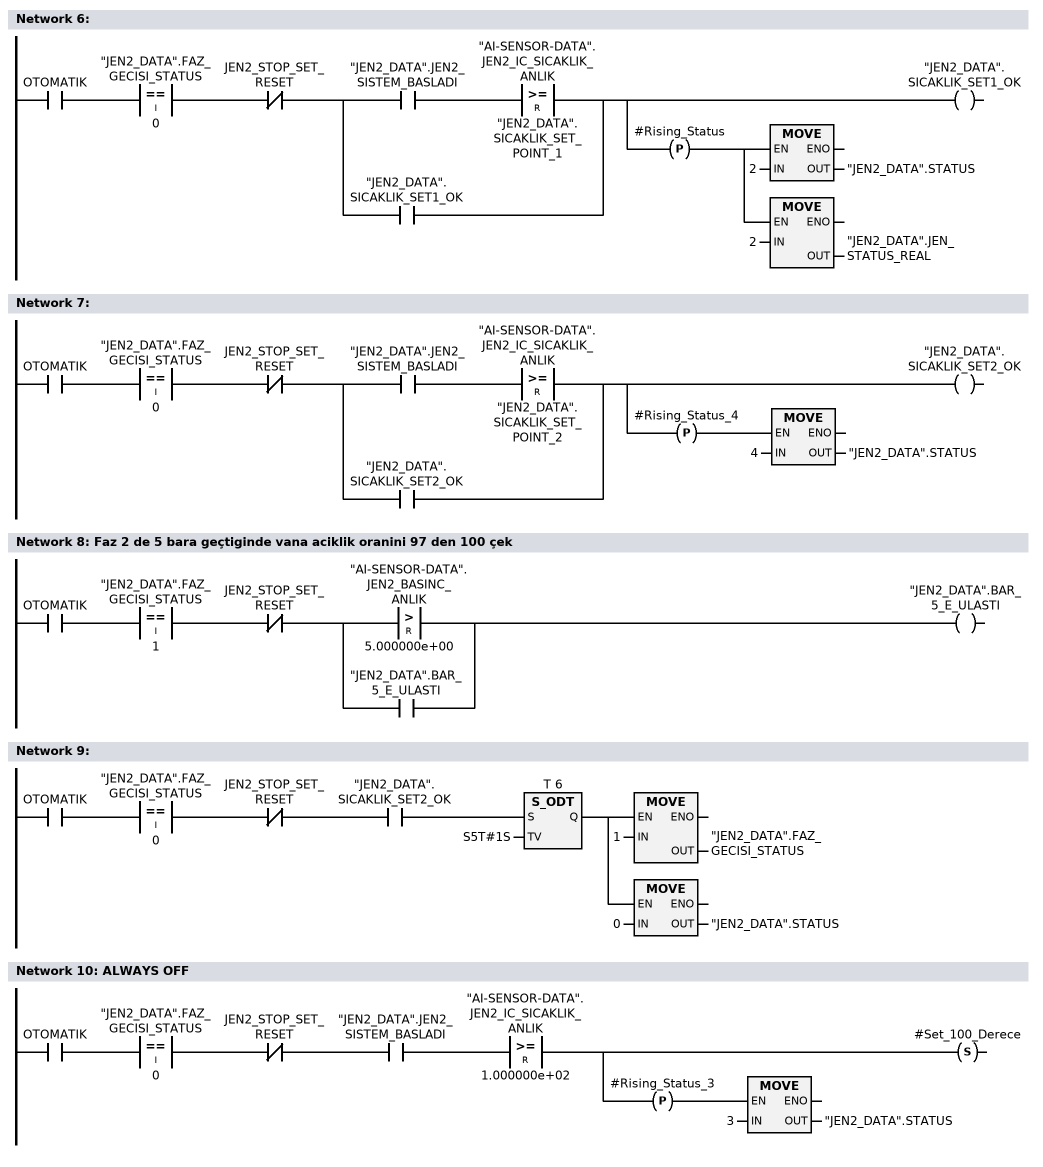
NETWORK
TITLE =
      A     "OTOMATIK";
      A(;
      L     "JEN2_DATA".FAZ_GECISI_STATUS;
      L     0;
      ==I;
      );
      AN    "JEN2_STOP_SET_RESET";
      A(;
      A     "JEN2_DATA".JEN2_SISTEM_BASLADI;
      A(;
      L     "AI-SENSOR-DATA".JEN2_IC_SICAKLIK_ANLIK;
      L     "JEN2_DATA".SICAKLIK_SET_POINT_1;
      >=R;
      );
      O     "JEN2_DATA".SICAKLIK_SET1_OK;
      );
      =     L 0.0;
      A     L 0.0;
      BLD   102;
      =     "JEN2_DATA".SICAKLIK_SET1_OK;
      A     L 0.0;
      FP    #Rising_Status;
      =     L 0.1;
      A     L 0.1;
      JNB   _006;
      L     2;
      T     "JEN2_DATA".STATUS;
_006: NOP   0;
      A     L 0.1;
      JNB   _007;
      L     2;
      T     "JEN2_DATA".JEN_STATUS_REAL;
_007: NOP   0;
NETWORK
TITLE =
      A     "OTOMATIK";
      A(;
      L     "JEN2_DATA".FAZ_GECISI_STATUS;
      L     0;
      ==I;
      );
      AN    "JEN2_STOP_SET_RESET";
      A(;
      A     "JEN2_DATA".JEN2_SISTEM_BASLADI;
      A(;
      L     "AI-SENSOR-DATA".JEN2_IC_SICAKLIK_ANLIK;
      L     "JEN2_DATA".SICAKLIK_SET_POINT_2;
      >=R;
      );
      O     "JEN2_DATA".SICAKLIK_SET2_OK;
      );
      =     L 0.0;
      A     L 0.0;
      BLD   102;
      =     "JEN2_DATA".SICAKLIK_SET2_OK;
      A     L 0.0;
      FP    #Rising_Status_4;
      JNB   _008;
      L     4;
      T     "JEN2_DATA".STATUS;
_008: NOP   0;
NETWORK
TITLE = Faz 2 de 5 bara geçtiginde vana aciklik oranini 97 den 100 çek
      A     "OTOMATIK";
      A(;
      L     "JEN2_DATA".FAZ_GECISI_STATUS;
      L     1;
      ==I;
      );
      AN    "JEN2_STOP_SET_RESET";
      A(;
      O(;
      L     "AI-SENSOR-DATA".JEN2_BASINC_ANLIK;
      L     5.000000e+00;
      >R;
      );
      O     "JEN2_DATA".BAR_5_E_ULASTI;
      );
      =     "JEN2_DATA".BAR_5_E_ULASTI;
NETWORK
TITLE =
//SET 2 SICAKLIGINDAN SONRA FAZ 2 E GEC
      A     "OTOMATIK";
      A(;
      L     "JEN2_DATA".FAZ_GECISI_STATUS;
      L     0;
      ==I;
      );
      AN    "JEN2_STOP_SET_RESET";
      A     "JEN2_DATA".SICAKLIK_SET2_OK;
      L     S5T#1S;
      SD    T 6;
      NOP   0;
      NOP   0;
      NOP   0;
      A     T 6;
      =     L 0.0;
      A     L 0.0;
      JNB   _009;
      L     1;
      T     "JEN2_DATA".FAZ_GECISI_STATUS;
_009: NOP   0;
      A     L 0.0;
      JNB   _00a;
      L     0;
      T     "JEN2_DATA".STATUS;
_00a: NOP   0;
NETWORK
TITLE = ALWAYS OFF
//Pompa 100 derecede duracak
      A     "OTOMATIK";
      A(;
      L     "JEN2_DATA".FAZ_GECISI_STATUS;
      L     0;
      ==I;
      );
      AN    "JEN2_STOP_SET_RESET";
      A     "JEN2_DATA".JEN2_SISTEM_BASLADI;
      A(;
      L     "AI-SENSOR-DATA".JEN2_IC_SICAKLIK_ANLIK;
      L     1.000000e+02;
      >=R;
      );
      =     L 0.0;
      A     L 0.0;
      BLD   102;
      S     #Set_100_Derece;
      A     L 0.0;
      FP    #Rising_Status_3;
      JNB   _00b;
      L     3;
      T     "JEN2_DATA".STATUS;
_00b: NOP   0;
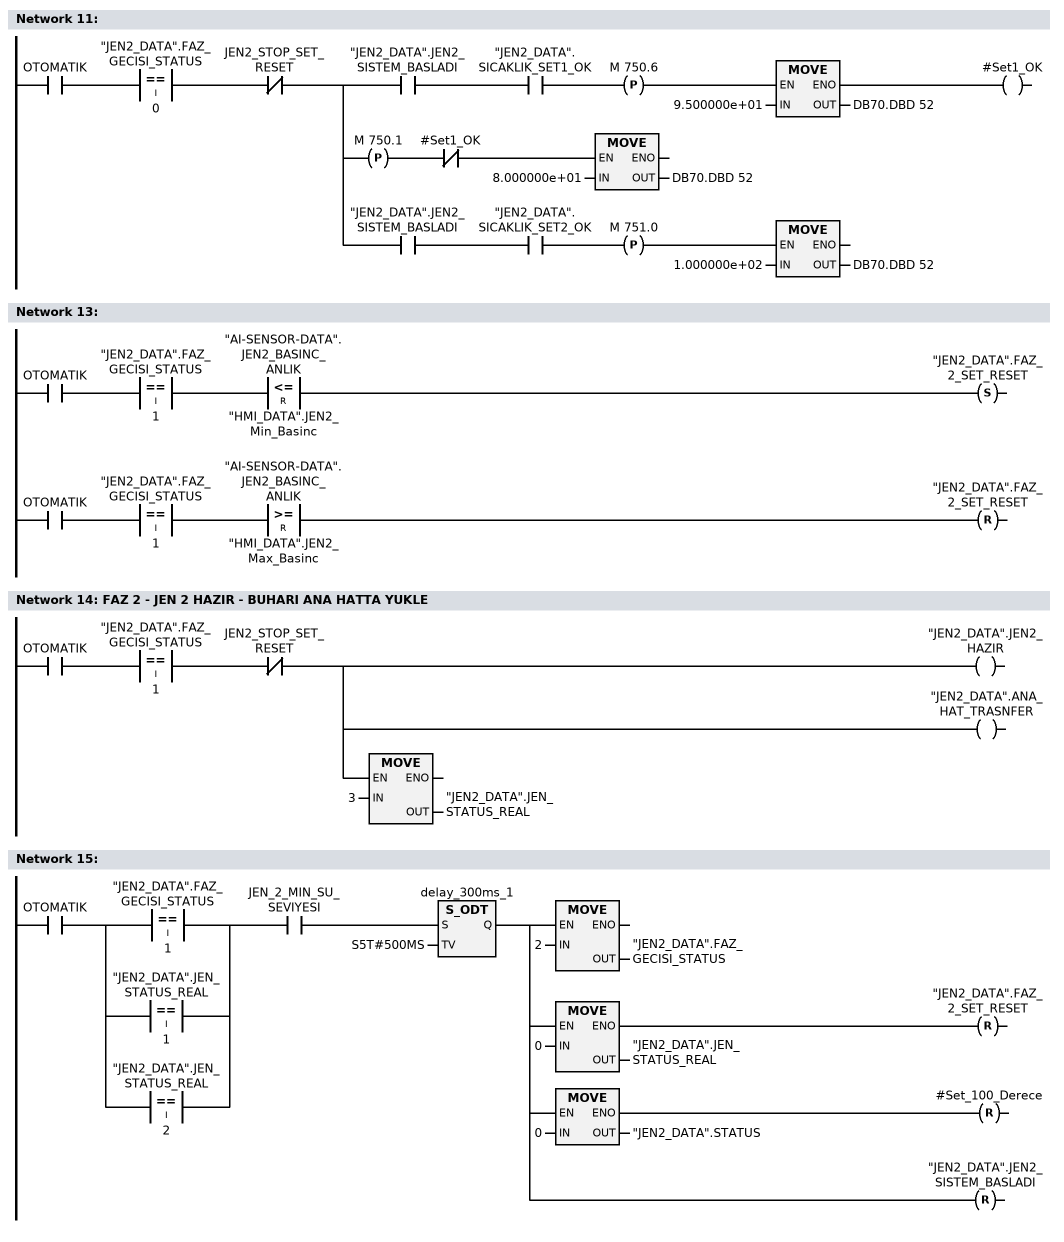
NETWORK
TITLE =
//-Sicaklik set 1 e geldiginde vana kapanma orani 5'e kadar düsüyor
//-Sicaklik set 2 e geldiginde vana kapanma orani 0'a kadar dusecek
      A     "OTOMATIK";
      A(;
      L     "JEN2_DATA".FAZ_GECISI_STATUS;
      L     0;
      ==I;
      );
      AN    "JEN2_STOP_SET_RESET";
      =     L 0.0;
      A     L 0.0;
      A     "JEN2_DATA".JEN2_SISTEM_BASLADI;
      A     "JEN2_DATA".SICAKLIK_SET1_OK;
      FP    M 750.6;
      JNB   _00c;
      L     9.500000e+01;
      T     DB70.DBD 52;
      SET;
      SAVE;
      CLR;
_00c: A     BR;
      =     #Set1_OK;
      A     L 0.0;
      FP    M 750.1;
      AN    #Set1_OK;
      JNB   _00d;
      L     8.000000e+01;
      T     DB70.DBD 52;
_00d: NOP   0;
      A     L 0.0;
      A     "JEN2_DATA".JEN2_SISTEM_BASLADI;
      A     "JEN2_DATA".SICAKLIK_SET2_OK;
      FP    M 751.0;
      JNB   _00e;
      L     1.000000e+02;
      T     DB70.DBD 52;
_00e: NOP   0;
NETWORK
TITLE =
NETWORK
TITLE =
//FAZ - 2 MODUNA GEÇ
//1-BURLOR VE POMPA 4.5-5.5 BAR ARASINDA ÇALISIP DURACAK
      A     "OTOMATIK";
      A(;
      L     "JEN2_DATA".FAZ_GECISI_STATUS;
      L     1;
      ==I;
      );
      A(;
      L     "AI-SENSOR-DATA".JEN2_BASINC_ANLIK;
      L     "HMI_DATA".JEN2_Min_Basinc;
      <=R;
      );
      S     "JEN2_DATA".FAZ_2_SET_RESET;
      A     "OTOMATIK";
      A(;
      L     "JEN2_DATA".FAZ_GECISI_STATUS;
      L     1;
      ==I;
      );
      A(;
      L     "AI-SENSOR-DATA".JEN2_BASINC_ANLIK;
      L     "HMI_DATA".JEN2_Max_Basinc;
      >=R;
      );
      R     "JEN2_DATA".FAZ_2_SET_RESET;
      NOP   0;
NETWORK
TITLE = FAZ 2 - JEN 2 HAZIR - BUHARI ANA HATTA YUKLE
      A     "OTOMATIK";
      A(;
      L     "JEN2_DATA".FAZ_GECISI_STATUS;
      L     1;
      ==I;
      );
      AN    "JEN2_STOP_SET_RESET";
      =     L 0.0;
      A     L 0.0;
      BLD   102;
      =     "JEN2_DATA".JEN2_HAZIR;
      A     L 0.0;
      BLD   102;
      =     "JEN2_DATA".ANA_HAT_TRASNFER;
      A     L 0.0;
      JNB   _00f;
      L     3;
      T     "JEN2_DATA".JEN_STATUS_REAL;
_00f: NOP   0;
NETWORK
TITLE =
//FAZ 3 - GUVENLIK ONLEMLERI 
//1- 6 bar asildiginda -ok
//2- Baca 180 dereceyi gecerse -ok
//3- Su miktari min altina duserse -ok
      A     "OTOMATIK";
      A(;
      O(;
      L     "JEN2_DATA".FAZ_GECISI_STATUS;
      L     1;
      ==I;
      );
      O(;
      L     "JEN2_DATA".JEN_STATUS_REAL;
      L     1;
      ==I;
      );
      O(;
      L     "JEN2_DATA".JEN_STATUS_REAL;
      L     2;
      ==I;
      );
      );
      A     "JEN_2_MIN_SU_SEVIYESI";
      L     S5T#500MS;
      SD    "delay_300ms_1";
      NOP   0;
      NOP   0;
      NOP   0;
      A     "delay_300ms_1";
      =     L 0.0;
      A     L 0.0;
      JNB   _010;
      L     2;
      T     "JEN2_DATA".FAZ_GECISI_STATUS;
_010: NOP   0;
      A     L 0.0;
      JNB   _011;
      L     0;
      T     "JEN2_DATA".JEN_STATUS_REAL;
      SET;
      SAVE;
      CLR;
_011: A     BR;
      R     "JEN2_DATA".FAZ_2_SET_RESET;
      A     L 0.0;
      JNB   _012;
      L     0;
      T     "JEN2_DATA".STATUS;
      SET;
      SAVE;
      CLR;
_012: A     BR;
      R     #Set_100_Derece;
      A     L 0.0;
      BLD   102;
      R     "JEN2_DATA".JEN2_SISTEM_BASLADI;
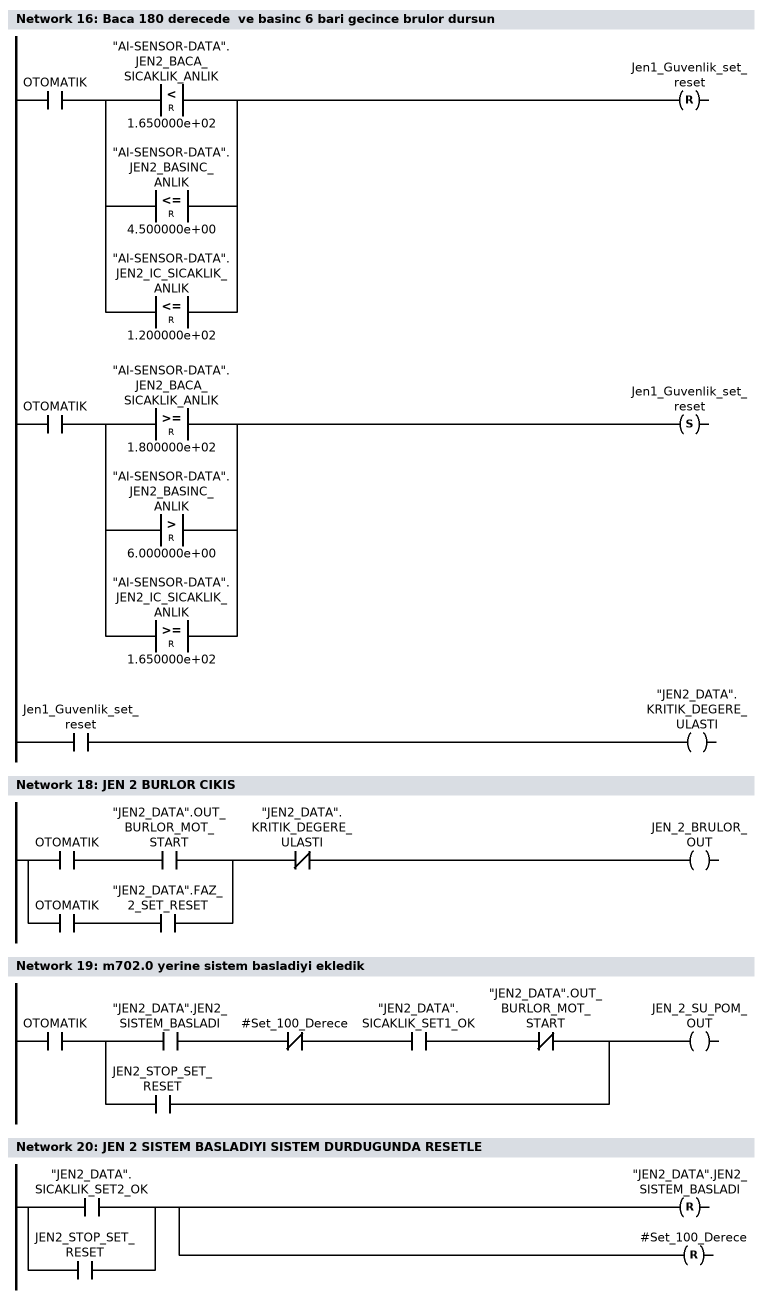
NETWORK
TITLE = Baca 180 derecede  ve basinc 6 bari gecince brulor dursun
      A     "OTOMATIK";
      A(;
      O(;
      L     "AI-SENSOR-DATA".JEN2_BACA_SICAKLIK_ANLIK;
      L     1.650000e+02;
      <R;
      );
      O(;
      L     "AI-SENSOR-DATA".JEN2_BASINC_ANLIK;
      L     4.500000e+00;
      <=R;
      );
      O(;
      L     "AI-SENSOR-DATA".JEN2_IC_SICAKLIK_ANLIK;
      L     1.200000e+02;
      <=R;
      );
      );
      R     "Jen1_Guvenlik_set_reset";
      A     "OTOMATIK";
      A(;
      O(;
      L     "AI-SENSOR-DATA".JEN2_BACA_SICAKLIK_ANLIK;
      L     1.800000e+02;
      >=R;
      );
      O(;
      L     "AI-SENSOR-DATA".JEN2_BASINC_ANLIK;
      L     6.000000e+00;
      >R;
      );
      O(;
      L     "AI-SENSOR-DATA".JEN2_IC_SICAKLIK_ANLIK;
      L     1.650000e+02;
      >=R;
      );
      );
      S     "Jen1_Guvenlik_set_reset";
      A     "Jen1_Guvenlik_set_reset";
      =     "JEN2_DATA".KRITIK_DEGERE_ULASTI;
NETWORK
TITLE =
NETWORK
TITLE = JEN 2 BURLOR CIKIS
      A(;
      A     "OTOMATIK";
      A     "JEN2_DATA".OUT_BURLOR_MOT_START;
      O;
      A     "OTOMATIK";
      A     "JEN2_DATA".FAZ_2_SET_RESET;
      );
      AN    "JEN2_DATA".KRITIK_DEGERE_ULASTI;
      =     "JEN_2_BRULOR_OUT";
NETWORK
TITLE = m702.0 yerine sistem basladiyi ekledik
      A     "OTOMATIK";
      A(;
      A     "JEN2_DATA".JEN2_SISTEM_BASLADI;
      AN    #Set_100_Derece;
      A     "JEN2_DATA".SICAKLIK_SET1_OK;
      AN    "JEN2_DATA".OUT_BURLOR_MOT_START;
      O     "JEN2_STOP_SET_RESET";
      );
      =     "JEN_2_SU_POM_OUT";
NETWORK
TITLE = JEN 2 SISTEM BASLADIYI SISTEM DURDUGUNDA RESETLE
      O     "JEN2_DATA".SICAKLIK_SET2_OK;
      O     "JEN2_STOP_SET_RESET";
      R     "JEN2_DATA".JEN2_SISTEM_BASLADI;
      R     #Set_100_Derece;
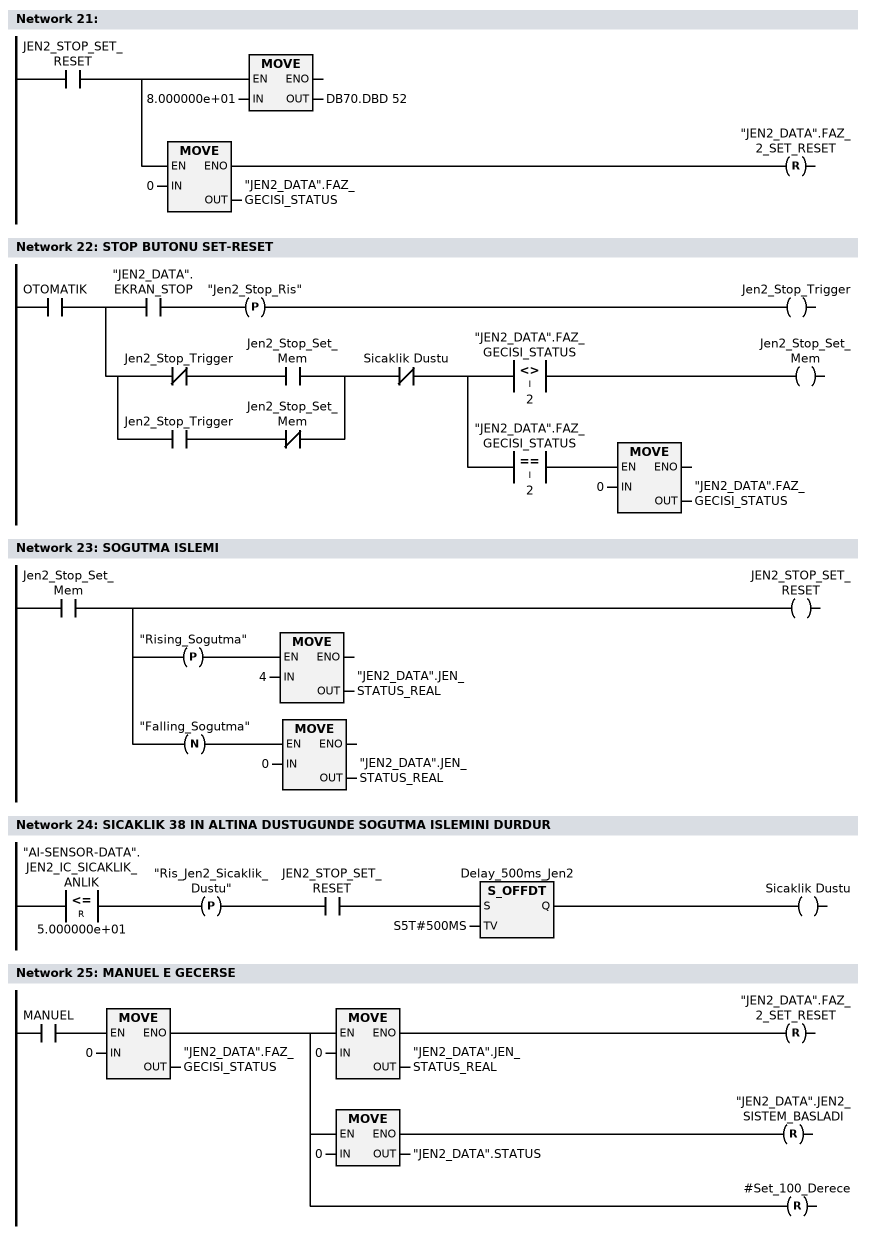
NETWORK
TITLE =
      A     "JEN2_STOP_SET_RESET";
      =     L 0.0;
      A     L 0.0;
      JNB   _013;
      L     8.000000e+01;
      T     DB70.DBD 52;
_013: NOP   0;
      A     L 0.0;
      JNB   _014;
      L     0;
      T     "JEN2_DATA".FAZ_GECISI_STATUS;
      SET;
      SAVE;
      CLR;
_014: A     BR;
      R     "JEN2_DATA".FAZ_2_SET_RESET;
NETWORK
TITLE = STOP BUTONU SET-RESET
      A     "OTOMATIK";
      =     L 0.0;
      A     L 0.0;
      A     "JEN2_DATA".EKRAN_STOP;
      FP    "Jen2_Stop_Ris";
      =     "Jen2_Stop_Trigger";
      A     L 0.0;
      A(;
      AN    "Jen2_Stop_Trigger";
      A     "Jen2_Stop_Set_Mem";
      O;
      A     "Jen2_Stop_Trigger";
      AN    "Jen2_Stop_Set_Mem";
      );
      AN    "Sicaklik Dustu";
      =     L 0.1;
      A     L 0.1;
      A(;
      L     "JEN2_DATA".FAZ_GECISI_STATUS;
      L     2;
      <>I;
      );
      =     "Jen2_Stop_Set_Mem";
      A     L 0.1;
      A(;
      L     "JEN2_DATA".FAZ_GECISI_STATUS;
      L     2;
      ==I;
      );
      JNB   _015;
      L     0;
      T     "JEN2_DATA".FAZ_GECISI_STATUS;
_015: NOP   0;
NETWORK
TITLE = SOGUTMA ISLEMI
      A     "Jen2_Stop_Set_Mem";
      =     L 0.0;
      A     L 0.0;
      BLD   102;
      =     "JEN2_STOP_SET_RESET";
      A     L 0.0;
      FP    "Rising_Sogutma";
      JNB   _016;
      L     4;
      T     "JEN2_DATA".JEN_STATUS_REAL;
_016: NOP   0;
      A     L 0.0;
      FN    "Falling_Sogutma";
      JNB   _017;
      L     0;
      T     "JEN2_DATA".JEN_STATUS_REAL;
_017: NOP   0;
NETWORK
TITLE = SICAKLIK 38 IN ALTINA DUSTUGUNDE SOGUTMA ISLEMINI DURDUR
      A(;
      L     "AI-SENSOR-DATA".JEN2_IC_SICAKLIK_ANLIK;
      L     5.000000e+01;
      <=R;
      );
      FP    "Ris_Jen2_Sicaklik_Dustu";
      A     "JEN2_STOP_SET_RESET";
      L     S5T#500MS;
      SF    "Delay_500ms_Jen2";
      NOP   0;
      NOP   0;
      NOP   0;
      A     "Delay_500ms_Jen2";
      =     "Sicaklik Dustu";
NETWORK
TITLE = MANUEL E GECERSE
      A     "MANUEL";
      JNB   _018;
      L     0;
      T     "JEN2_DATA".FAZ_GECISI_STATUS;
      SET;
      SAVE;
      CLR;
_018: A     BR;
      =     L 0.0;
      A     L 0.0;
      JNB   _019;
      L     0;
      T     "JEN2_DATA".JEN_STATUS_REAL;
      SET;
      SAVE;
      CLR;
_019: A     BR;
      R     "JEN2_DATA".FAZ_2_SET_RESET;
      A     L 0.0;
      JNB   _01a;
      L     0;
      T     "JEN2_DATA".STATUS;
      SET;
      SAVE;
      CLR;
_01a: A     BR;
      R     "JEN2_DATA".JEN2_SISTEM_BASLADI;
      A     L 0.0;
      BLD   102;
      R     #Set_100_Derece;
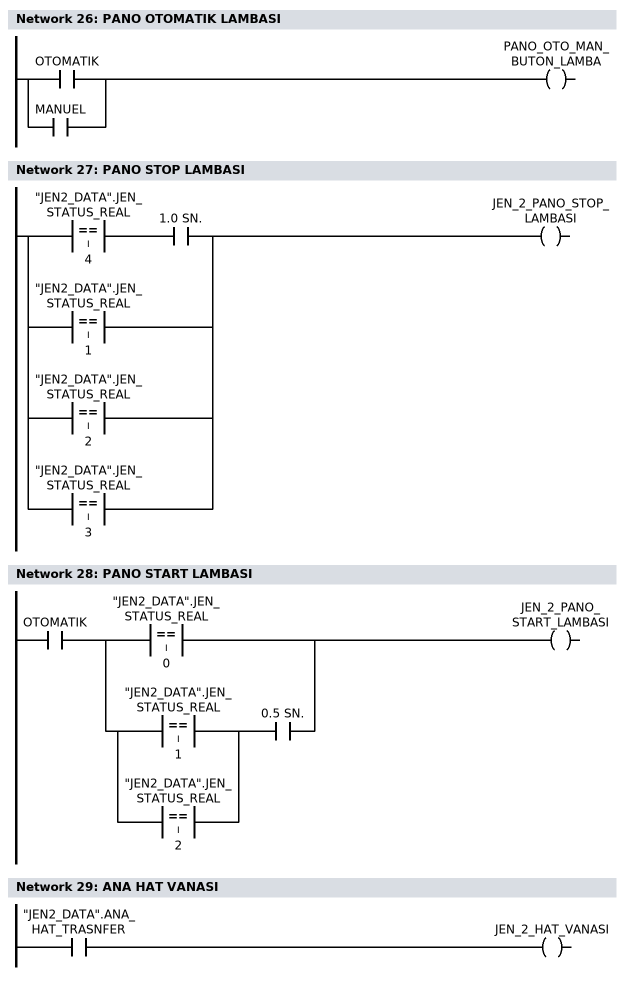
NETWORK
TITLE = PANO OTOMATIK LAMBASI
      O     "OTOMATIK";
      O     "MANUEL";
      =     "PANO_OTO_MAN_BUTON_LAMBA";
NETWORK
TITLE = PANO STOP LAMBASI
//1- Buhar hazýrlaniyor
//2- set 1 e ulasti
//3- Basinci Stabil tutma
//4- Sogutma
      A(;
      L     "JEN2_DATA".JEN_STATUS_REAL;
      L     4;
      ==I;
      );
      A     "1.0 SN.";
      O(;
      L     "JEN2_DATA".JEN_STATUS_REAL;
      L     1;
      ==I;
      );
      O(;
      L     "JEN2_DATA".JEN_STATUS_REAL;
      L     2;
      ==I;
      );
      O(;
      L     "JEN2_DATA".JEN_STATUS_REAL;
      L     3;
      ==I;
      );
      =     "JEN_2_PANO_STOP_LAMBASI";
NETWORK
TITLE = PANO START LAMBASI
      A     "OTOMATIK";
      A(;
      O(;
      L     "JEN2_DATA".JEN_STATUS_REAL;
      L     0;
      ==I;
      );
      O;
      A(;
      O(;
      L     "JEN2_DATA".JEN_STATUS_REAL;
      L     1;
      ==I;
      );
      O(;
      L     "JEN2_DATA".JEN_STATUS_REAL;
      L     2;
      ==I;
      );
      );
      A     "0.5 SN.";
      );
      =     "JEN_2_PANO_START_LAMBASI";
NETWORK
TITLE = ANA HAT VANASI 
      A     "JEN2_DATA".ANA_HAT_TRASNFER;
      =     "JEN_2_HAT_VANASI";
END_FUNCTION_BLOCK

FUNCTION "TIME_UNSCALE" : VOID	// FC 1
VERSION : 0.0
VAR_INPUT
  iTimeET : TIME ;
  iIstenileSure : S5TIME ;
END_VAR
VAR_OUTPUT
  oOUT : DINT ;
END_VAR
VAR_TEMP
  vTemp : DINT ;
  vValue : DINT ;
  vValue2 : DINT ;
  vIstenilenTime : TIME ;
  vIstenilenDint : DINT ;
END_VAR
BEGIN
// body was compiled from an SCL source; compiled code not shown
END_FUNCTION

FUNCTION "O.Vana_AciklikHesaplama" : VOID	// FC 2
VERSION : 0.1
VAR_INPUT
  IlkAciklikDegeri : REAL ;
  KademeliAcikDegeri : REAL ;
END_VAR
VAR_OUTPUT
  oKademe_1 : REAL ;
  oKademe_2 : REAL ;
  oKademe_3 : REAL ;
  oKademe_4 : REAL ;
  oKademe_5 : REAL ;
  oKademe_6 : REAL ;
  oKademe_7 : REAL ;
END_VAR
VAR_TEMP
  tKademe : STRUCT
   Iki : REAL ;
   Uc : REAL ;
   Dort : REAL ;
   Bes : REAL ;
   Alti : REAL ;
   Yedi : REAL ;
  END_STRUCT ;
  tCheck_Kademe5 : BOOL ;
  tCheck_Kademe6 : BOOL ;
  tCheck_Kademe7 : BOOL ;
END_VAR
BEGIN
NETWORK
TITLE =
//------------------------
// kademe 1
      L     #IlkAciklikDegeri;
      T     #oKademe_1;
//------------------------
// kademe 2
      L     #IlkAciklikDegeri;
      L     #KademeliAcikDegeri;
      +R;
      T     #tKademe.Iki;
      L     #tKademe.Iki;
      T     #oKademe_2;
//-----------------------
// kademe 3
      L     #KademeliAcikDegeri;
      L     #tKademe.Iki;
      +R;
      T     #tKademe.Uc;
      L     #tKademe.Uc;
      T     #oKademe_3;
//-----------------------
// kademe 4
      L     #KademeliAcikDegeri;
      L     #tKademe.Uc;
      +R;
      T     #tKademe.Dort;
      L     #tKademe.Dort;
      T     #oKademe_4;
//-----------------------
// kademe 5
      L     #KademeliAcikDegeri;
      L     #tKademe.Dort;
      +R;
      T     #tKademe.Bes;
      L     #tKademe.Bes;
      L     6.000000e+01;
      >R;
      =     #tCheck_Kademe5;
      A     #tCheck_Kademe5;
      JNB   j005;
      L     6.000000e+01;
      T     #tKademe.Bes;
j005: NOP   0;
      L     #tKademe.Bes;
      T     #oKademe_5;
//-----------------------
// kademe 6
      L     #KademeliAcikDegeri;
      L     #tKademe.Bes;
      +R;
      T     #tKademe.Alti;
      L     #tKademe.Alti;
      L     6.000000e+01;
      >R;
      =     #tCheck_Kademe6;
      A     #tCheck_Kademe6;
      JNB   j006;
      L     6.000000e+01;
      T     #tKademe.Alti;
j006: NOP   0;
      L     #tKademe.Alti;
      T     #oKademe_6;
//-----------------------
// kademe 7
      L     #KademeliAcikDegeri;
      L     #tKademe.Alti;
      +R;
      T     #tKademe.Yedi;
      L     #tKademe.Yedi;
      L     6.000000e+01;
      >R;
      =     #tCheck_Kademe7;
      A     #tCheck_Kademe7;
      JNB   j007;
      L     6.000000e+01;
      T     #tKademe.Yedi;
j007: NOP   0;
      L     #tKademe.Yedi;
      T     #oKademe_7;
NETWORK
TITLE =
END_FUNCTION

FUNCTION "IntToS5Time" : VOID	// FC 10
VERSION : 0.0
VAR_INPUT
  Saat : INT ;
  Dakika : INT ;
END_VAR
VAR_OUTPUT
  HesaplananSure_S5TIME : S5TIME ;
END_VAR
VAR_TEMP
  tSaat_Dint : DINT ;
  tHesaplananSaat : DINT ;
  tDakika_Dint : DINT ;
  tHesaplananDakika : DINT ;
  tHesaplnananSure_Dint : DINT ;
  tHesaplananSure_Time : TIME ;
END_VAR
BEGIN
// body was compiled from an SCL source; compiled code not shown
END_FUNCTION

// FC 33: know-how protected block, not included

// FC 40: know-how protected block, not included

// FC 105: know-how protected block, not included

// FC 106: know-how protected block, not included

DATA_BLOCK "AI-SENSOR-DATA"	// DB 1
VERSION : 0.1
  STRUCT
   JEN1_BASINC_ANLIK : REAL ;
   JEN2_BASINC_ANLIK : REAL ;
   JEN1_BASINC_RET_VAL : WORD ;
   JEN2_BASINC_RET_VAL : WORD ;
   JEN1_IC_SICAKLIK_ANLIK : REAL ;
   JEN2_IC_SICAKLIK_ANLIK : REAL ;
   JEN1_IC_SICAKLIK_RET_VAL : WORD ;
   JEN2_IC_SICAKLIK_RET_VAL : WORD ;
   JEN1_BACA_SICAKLIK_ANLIK : REAL ;
   JEN2_BACA_SICAKLIK_ANLIK : REAL ;
   JEN1_BACA_SICAKLIK_RET_V : WORD ;
   JEN2_BACA_SICAKLIK_RET_V : WORD ;
   HAT_BASINCI_RET_V : WORD ;
   HAT_BASINCI_ANLIK : REAL ;
   HAVA_BASINCI_RET_V : WORD ;
   HAVA_BASINCI_ANLIK : REAL ;
   HAT_BASINCI_YETERLI : BOOL ;
  END_STRUCT ;	
BEGIN
END_DATA_BLOCK

DATA_BLOCK "ORTAK_DATA"	// DB 2
VERSION : 0.1
  STRUCT
   JEN_EMNIYET_BASINCI : REAL ;
   JEN_EMNIYET_SICAKLIGI : REAL ;
   OTO_EMNIYET_BASINCI : REAL ;
   OTO_EMNIYET_SICAKLIGI : REAL ;
   OTO_ISLEM_BITTI_VANA_AC : BOOL ;
   OTO_JEN_DURDU : REAL ;
  END_STRUCT ;	
BEGIN
END_DATA_BLOCK

DATA_BLOCK "TIME_OTO_1_DB"	// DB 5
AUTHOR : SIMATIC
FAMILY : IEC_TC
VERSION : 0.0
"TON"
BEGIN
END_DATA_BLOCK

DATA_BLOCK "TIME_OTO_2_DB"	// DB 6
AUTHOR : SIMATIC
FAMILY : IEC_TC
VERSION : 0.0
"TON"
BEGIN
END_DATA_BLOCK

DATA_BLOCK "TIME_OTO_1_PROSES_DB"	// DB 7
AUTHOR : SIMATIC
FAMILY : IEC_TC
VERSION : 0.0
"TON"
BEGIN
END_DATA_BLOCK

DATA_BLOCK "TIME_OTO_2_PROSES_DB"	// DB 8
AUTHOR : SIMATIC
FAMILY : IEC_TC
VERSION : 0.0
"TON"
BEGIN
END_DATA_BLOCK

DATA_BLOCK DB 9
AUTHOR : SIMATIC
FAMILY : IEC_TC
VERSION : 0.0
"TON"
BEGIN
END_DATA_BLOCK

DATA_BLOCK DB 10
AUTHOR : SIMATIC
FAMILY : IEC_TC
VERSION : 0.0
"TON"
BEGIN
END_DATA_BLOCK

DATA_BLOCK "SURELER_DB"	// DB 14
VERSION : 0.0
"SURELER"
BEGIN
END_DATA_BLOCK

DATA_BLOCK "SAFETY_DB"	// DB 15
VERSION : 0.0
"SAFETY"
BEGIN
END_DATA_BLOCK

DATA_BLOCK "KAZAN1_DATA"	// DB 17
VERSION : 0.1
  STRUCT
   IN_STATUS : INT ;
   IN_JEN_OK : BOOL ;
   IN_DIGER_KAZ_TRANS_HAZIR : BOOL ;
   IN_PISIM_SURESI : S5TIME ;
   IN_SCALE_BASINC_PER : INT ;
   IN_SET_BASINC : REAL ;
   IN_DIGER_KAZAN_BASINCI : REAL ;
   O_PID_MAN_ON : BOOL ;
   O_PID_MAN : REAL ;
   O_TRANSFER_YAPILIYOR : BOOL ;
   O_SCALE_BASINC_RET_VAL : WORD ;
   O_SCALE_BASINC_OUT : REAL ;
   O_TRANSFERE_HAZIR : BOOL ;
   O_SCALE_SICAKLIK_RET_VAL : WORD ;
   O_SCALE_SICAKLIK_OUT : REAL ;
   IN_SCALE_SICAKLIK_PER : INT ;
   O_KAZAN_BOSALTIMDA : BOOL ;
   IN_DIGER_KAZ_BOSALTIMDA : BOOL ;
   IN_DIGER_KAZ_TRANSFERDE : BOOL ;
   O_PISIM_BASLADI : BOOL ;
   PISIM_GECEN_SURE_TIME : TIME ;
   PISIM_GECEN_SURE_DINT : DINT ;
   PROSES_SURESI_TIME : TIME ;
   PROSES_SURESI_DINT : DINT ;
   BEKLEME_SURESI_TIME : TIME ;
   BEKLEME_SURESI_DINT : DINT ;
  END_STRUCT ;	
BEGIN
END_DATA_BLOCK

DATA_BLOCK "KAZAN2_DATA"	// DB 18
VERSION : 0.1
  STRUCT
   IN_STATUS : INT ;
   IN_JEN_OK : BOOL ;
   IN_DIGER_KAZ_TRANS_HAZIR : BOOL ;
   IN_PISIM_SURESI : S5TIME ;
   IN_SCALE_BASINC_PER : INT ;
   IN_SET_BASINC : REAL ;
   IN_DIGER_KAZAN_BASINCI : REAL ;
   O_PID_MAN_ON : BOOL ;
   O_PID_MAN : REAL ;
   O_TRANSFER_YAPILIYOR : BOOL ;
   O_SCALE_BASINC_RET_VAL : WORD ;
   O_SCALE_BASINC_OUT : REAL ;
   O_TRANSFERE_HAZIR : BOOL ;
   O_SCALE_SICAKLIK_RET_VAL : WORD ;
   O_SCALE_SICAKLIK_OUT : REAL ;
   IN_SCALE_SICAKLIK_PER : INT ;
   O_KAZAN_BOSALTIMDA : BOOL ;
   IN_DIGER_KAZ_BOSALTIMDA : BOOL ;
   IN_DIGER_KAZ_TRANSFERDE : BOOL ;
   O_PISIM_BASLADI : BOOL ;
   PISIM_GECEN_SURE_TIME : TIME ;
   PISIM_GECEN_SURE_DINT : DINT ;
   PROSES_SURESI_TIM : TIME ;
   PROSES_SURESI_DINT : DINT ;
   BEKLEME_SURESI_TIME : TIME ;
   BEKLEME_SURESI_DINT : DINT ;
  END_STRUCT ;	
BEGIN
END_DATA_BLOCK

DATA_BLOCK "JEN1_DATA"	// DB 19
VERSION : 0.1
  STRUCT
   BASINC_SET_POINT : REAL ;
   STATUS : INT ;
   SICAKLIK_SET_POINT_1 : REAL ;
   SICAKLIK_SET_POINT_2 : REAL ;
   SISTEM_BASLADI : BOOL ;
   EKRAN_START : BOOL ;
   EKRAN_STOP : BOOL ;
   OUT_BURLOR_MOT_START : BOOL ;
   SICAKLIK_SET1_OK : BOOL ;
   SICAKLIK_SET2_OK : BOOL ;
   OUT_PID_START : BOOL ;
   FAZ_GECISI_STATUS : INT ;
   FAZ_2_SET_RESET : BOOL ;
   BAR_5_E_ULASTI : BOOL ;
   JEN1_HAZIR : BOOL ;
   ANA_HAT_TRASFER_HAZIR : BOOL ;
   JEN_STATUS_REAL : INT ;
   STOP_SET_RESET : BOOL ;
   CALISMA_SURESI_TIME : TIME ;
   CALISMA_SURESI_DINT : DINT ;
   KRITIK_DEGERLERE_ULASTI : BOOL ;	//180 derece baca-6 bari gecti- 165 ic sicaklik
   CALISMA_SURESI_EKRAN : DINT ;
   SET2_DEGERINE_ULASMADI : BOOL ;
  END_STRUCT ;	
BEGIN
END_DATA_BLOCK

DATA_BLOCK "JEN2_DATA"	// DB 20
VERSION : 0.1
  STRUCT
   BASINC_SET_POINT : REAL ;
   STATUS : INT ;
   SICAKLIK_SET_POINT_1 : REAL ;
   SICAKLIK_SET_POINT_2 : REAL ;
   JEN2_SISTEM_BASLADI : BOOL ;
   EKRAN_START : BOOL ;
   EKRAN_STOP : BOOL ;
   OUT_BURLOR_MOT_START : BOOL ;
   SICAKLIK_SET1_OK : BOOL ;
   SICAKLIK_SET2_OK : BOOL ;
   OUT_PID_START : BOOL ;
   FAZ_GECISI_STATUS : INT ;
   FAZ_2_SET_RESET : BOOL ;
   BAR_5_E_ULASTI : BOOL ;
   JEN2_HAZIR : BOOL ;
   ANA_HAT_TRASNFER : BOOL ;
   JEN_STATUS_REAL : INT ;
   STOP_SET_RESET : BOOL ;
   CALISMA_SURESI_TIME : TIME ;
   CALISMA_SURESI_DINT : DINT ;
   KRITIK_DEGERE_ULASTI : BOOL ;	//Baca 180 derecede-6 bari gecti-165 ic sicaklik
   CALISMA_SURESI_EKRAN : DINT ;
  END_STRUCT ;	
BEGIN
END_DATA_BLOCK

DATA_BLOCK "JEN1_PID_DATA"	// DB 21
VERSION : 0.1
  STRUCT
   TCONT_C_LMN : REAL ;
   TCONT_C_LMN_PER : INT ;
  END_STRUCT ;	
BEGIN
END_DATA_BLOCK

DATA_BLOCK "JEN2_PID_DATA"	// DB 22
VERSION : 0.1
  STRUCT
   TCONT_C_LMN : REAL ;
   TCONT_C_LMN_PER : INT ;
  END_STRUCT ;	
BEGIN
END_DATA_BLOCK

DATA_BLOCK "KAZAN1_PID_DATA"	// DB 23
VERSION : 0.1
  STRUCT
   TCONT_LMN_PER : INT ;
   TCONT_LMN : REAL ;
  END_STRUCT ;	
BEGIN
END_DATA_BLOCK

DATA_BLOCK "KAZAN2_PID_DATA"	// DB 24
VERSION : 0.1
  STRUCT
   TCONT_LMN_PER : INT ;
   TCONT_LMN : REAL ;
  END_STRUCT ;	
BEGIN
END_DATA_BLOCK

DATA_BLOCK DB 50
AUTHOR : SIMATIC
FAMILY : ICONT
VERSION : 0.0
"CONT_C"
BEGIN
END_DATA_BLOCK

DATA_BLOCK "JEN2_KONTROL_BLOGU_DB"	// DB 51
VERSION : 0.0
"JEN2_PID_KONTROL"
BEGIN
END_DATA_BLOCK

DATA_BLOCK DB 52
VERSION : 0.0
"JEN1_PID_KONTROL"
BEGIN
END_DATA_BLOCK

DATA_BLOCK "JEN_1_PID_DB"	// DB 69
AUTHOR : SIMATIC
FAMILY : CONTROL
VERSION : 0.0
"TCONT_CP"
BEGIN
END_DATA_BLOCK

DATA_BLOCK "JEN_2_PID_DB"	// DB 70
AUTHOR : SIMATIC
FAMILY : CONTROL
VERSION : 0.0
"TCONT_CP"
BEGIN
END_DATA_BLOCK

DATA_BLOCK "OTOKLAV_1_DB"	// DB 94
VERSION : 0.0
"KAZAN_1_KONTROL"
BEGIN
END_DATA_BLOCK

DATA_BLOCK "OTOKLAV_2_DB"	// DB 95
VERSION : 0.0
"KAZAN_2_KONTROL"
BEGIN
END_DATA_BLOCK

DATA_BLOCK "FB98_DB"	// DB 98
VERSION : 0.0
"JEN1_KONTROL_BLOGU"
BEGIN
END_DATA_BLOCK

DATA_BLOCK "FB99_DB"	// DB 99
VERSION : 0.0
"JEN2_KONTROL_BLOGU"
BEGIN
END_DATA_BLOCK

DATA_BLOCK "HMI_DATA"	// DB 100
VERSION : 0.1
  STRUCT
   JEN1_Min_Basinc : REAL  := 5.000000e+000;	//Jenerator 1 min otomatik sekans basinci
   JEN1_Max_Basinc : REAL  := 5.500000e+000;	//Jenerator 1 max otomatik sekans basinci
   JEN2_Min_Basinc : REAL  := 5.000000e+000;	//Jenerator 2 min otomatik sekans basinci
   JEN2_Max_Basinc : REAL  := 5.500000e+000;	//Jenerator 2 max otomatik sekans basinci
   OTOKLAV_First_Oran : REAL  := 2.000000e+001;	//Otoklav oransal vana otomatik sekans ilk acilis orani
   OTOKLAV_Kademeli_Artis : REAL  := 5.000000e+000;	//Otoklav oransal vana kademeli artis katsayisi
   Otoklav_1_TimeData : STRUCT 	//Otoklav 1 hmi süre bilgisi
    Hours : INT ;	//Istenen calisma saati
    Minutes : INT  := 30;	//Istenen calisma dakikasi
    Second : INT ;	//Istenen calisma saniyesi
   END_STRUCT ;
   Otoklav_2_TimeData : STRUCT 	//Otoklav 2 hmi süre bilgisi
    Hours : INT ;	//Istenen calisma saati
    Minutes : INT  := 30;	//Istenen calisma dakikasi
    Second : INT ;	//Istenen calisma saniyesi
   END_STRUCT ;
  END_STRUCT ;	
BEGIN
   JEN1_Min_Basinc := 5.000000e+00;
   JEN1_Max_Basinc := 5.500000e+00;
   JEN2_Min_Basinc := 5.000000e+00;
   JEN2_Max_Basinc := 5.500000e+00;
   Otoklav_1_TimeData.Minutes := 30;
   Otoklav_2_TimeData.Minutes := 30;
END_DATA_BLOCK

DATA_BLOCK DB 120
VERSION : 0.0
"KAZAN_ORTAK"
BEGIN
END_DATA_BLOCK

DATA_BLOCK "KAZAN_1_PID_DB"	// DB 130
AUTHOR : SIMATIC
FAMILY : CONTROL
VERSION : 0.0
"TCONT_CP"
BEGIN
END_DATA_BLOCK

DATA_BLOCK DB 131
VERSION : 0.0
"KAZAN_1_PID_KONTROL"
BEGIN
END_DATA_BLOCK

DATA_BLOCK DB 132
VERSION : 0.0
"KAZAN_2_PID_KONTROL"
BEGIN
END_DATA_BLOCK

DATA_BLOCK DB 230
VERSION : 0.0
"KAZAN_ORTAK"
BEGIN
END_DATA_BLOCK

DATA_BLOCK "KAZAN_2_PID_DATA"	// DB 231
AUTHOR : SIMATIC
FAMILY : CONTROL
VERSION : 0.0
"TCONT_CP"
BEGIN
END_DATA_BLOCK

DATA_BLOCK DB 232
VERSION : 0.0
"TEST_BLOGU"
BEGIN
END_DATA_BLOCK

ORGANIZATION_BLOCK OB 1
TITLE = "Main Program Sweep (Cycle)"
VERSION : 0.1
VAR_TEMP
  OB1_EV_CLASS : BYTE ;	//Bits 0-3 = 1 (Coming event), Bits 4-7 = 1 (Event class 1)
  OB1_SCAN_1 : BYTE ;	//1 (Cold restart scan 1 of OB 1), 3 (Scan 2-n of OB 1)
  OB1_PRIORITY : BYTE ;	//Priority of OB Execution
  OB1_OB_NUMBR : BYTE ;	//1 (Organization block 1, OB1)
  OB1_RESERVED_1 : BYTE ;	//Reserved for system
  OB1_RESERVED_2 : BYTE ;	//Reserved for system
  OB1_PREV_CYCLE : INT ;	//Cycle time of previous OB1 scan (milliseconds)
  OB1_MIN_CYCLE : INT ;	//Minimum cycle time of OB1 (milliseconds)
  OB1_MAX_CYCLE : INT ;	//Maximum cycle time of OB1 (milliseconds)
  OB1_DATE_TIME : DATE_AND_TIME ;	//Date and time OB1 started
END_VAR
BEGIN
NETWORK
TITLE = ALWAYS OFF
      UC    "MAINBLOCK";
NETWORK
TITLE = HAVA VE HAT BASINCI
      CALL  "SCALE" (
           $1                       := P#P 292.0,
           $2                       := L#1092616192,
           $3                       := L#0,
           $4                       := "ALWAYS OFF",
           $5                       := "AI-SENSOR-DATA".HAT_BASINCI_RET_V,
           $6                       := "AI-SENSOR-DATA".HAT_BASINCI_ANLIK);
      CALL  "SCALE" (
           $1                       := P#P 294.0,
           $2                       := L#1092616192,
           $3                       := L#0,
           $4                       := "ALWAYS OFF",
           $5                       := "AI-SENSOR-DATA".HAVA_BASINCI_RET_V,
           $6                       := "AI-SENSOR-DATA".HAVA_BASINCI_ANLIK);
NETWORK
TITLE = ACIKLAMALAR
//FB98 - JEN 1 KONTROL BLOGU
//FB99 - JEN 2 KONTROL BLOGU
//FB49 - JEN 1 PID KONTROL - PID BLOKLARI
//FB50 - JEN 2 PID KONTROL - PID BLOKLARI
//FB94 - KAZAN 1 KONTROL BLOGU - KAZAN 1 ILE ILGILI KONTROLLER
//FB95 - KAZAN 2 KONTROL BLOGU - KAZAN 2 ILE ILGILI KONTROLLER
//FB47 - KAZAN 1 PID KONTROL
//FB48 - KAZAN 2 PID KONTROL
//FB3 - SURELER - KAZAN1,KAZAN2, JEN1, JEN2 ILE ILGILI TUM SURELER BURADA TUTULUR
//FB2 - SAFETY
//      1)JEN1, JEN2 KRITIK SU SEVIYE MIKTARLARI
//      2)HAVA BASINCI KONTROLU
//      3)JENERATOR IS BITIMINDE BORUDA KALAN BUHARIN TAHLIYESI
//FB1 - MAINBLOCK  
//      1)ÇALISACAK TUM BLOKLAR BURADA CAGRILIR
//      2)AYRICA HAVA VE HAT BASINCI DONUSUMLARI BURADADIR
//FB5 - TEST BLOGU - PROSESIN DEVREYE ALINAMADAN ONCEKI TEST ISLEMLERININ GERCEKLESTIGI
//      BLOKTUR.
END_ORGANIZATION_BLOCK

ORGANIZATION_BLOCK "PID BLOCK"	// OB 35
TITLE = "Cyclic Interrupt"
VERSION : 0.1
VAR_TEMP
  OB35_EV_CLASS : BYTE ;	//Bits 0-3 = 1 (Coming event), Bits 4-7 = 1 (Event class 1)
  OB35_STRT_INF : BYTE ;	//16#36 (OB 35 has started)
  OB35_PRIORITY : BYTE ;	//Priority of OB Execution
  OB35_OB_NUMBR : BYTE ;	//35 (Organization block 35, OB35)
  OB35_RESERVED_1 : BYTE ;	//Reserved for system
  OB35_RESERVED_2 : BYTE ;	//Reserved for system
  OB35_PHASE_OFFSET : WORD ;	//Phase offset (msec)
  OB35_RESERVED_3 : INT ;	//Reserved for system
  OB35_EXC_FREQ : INT ;	//Frequency of execution (msec)
  OB35_DATE_TIME : DATE_AND_TIME ;	//Date and time OB35 started
END_VAR
BEGIN
NETWORK
TITLE =
      CALL  "JEN1_PID_KONTROL" , DB 52;
      CALL  "JEN2_PID_KONTROL" , "JEN2_KONTROL_BLOGU_DB";
NETWORK
TITLE =
      CALL  "KAZAN_1_PID_KONTROL" , DB 131;
      CALL  "KAZAN_2_PID_KONTROL" , DB 132;
END_ORGANIZATION_BLOCK

ORGANIZATION_BLOCK "ZAMANHATASI"	// OB 80
TITLE = "Cycle Time Fault"
VERSION : 0.1
VAR_TEMP
  OB80_EV_CLASS : BYTE ;	//16#35, Event class 3, Entering event state, Internal fault event
  OB80_FLT_ID : BYTE ;	//16#XX, Fault identifcation code
  OB80_PRIORITY : BYTE ;	//Priority of OB Execution
  OB80_OB_NUMBR : BYTE ;	//80 (Organization block 80, OB80)
  OB80_RESERVED_1 : BYTE ;	//Reserved for system
  OB80_RESERVED_2 : BYTE ;	//Reserved for system
  OB80_ERROR_INFO : WORD ;	//Error information on event
  OB80_ERR_EV_CLASS : BYTE ;	//Class of event causing error
  OB80_ERR_EV_NUM : BYTE ;	//Number of event causing error
  OB80_OB_PRIORITY : BYTE ;	//Priority of OB causing error
  OB80_OB_NUM : BYTE ;	//Number of OB causing error
  OB80_DATE_TIME : DATE_AND_TIME ;	//Date and time OB80 started
END_VAR
BEGIN
// (block stored without names or comments; labels and parameter names are numbered)
END_ORGANIZATION_BLOCK

ORGANIZATION_BLOCK "GERILIMHATASI"	// OB 81
TITLE = "Power Supply Fault"
VERSION : 0.1
VAR_TEMP
  OB81_EV_CLASS : BYTE ;	//16#39, Event class 3, Entering event state, Internal fault event
  OB81_FLT_ID : BYTE ;	//16#XX, Fault identifcation code
  OB81_PRIORITY : BYTE ;	//Priority of OB Execution
  OB81_OB_NUMBR : BYTE ;	//81 (Organization block 81, OB81)
  OB81_RESERVED_1 : BYTE ;	//Reserved for system
  OB81_RESERVED_2 : BYTE ;	//Reserved for system
  OB81_RACK_CPU : WORD ;	//see online help (F1)
  OB81_RESERVED_3 : BYTE ;	//Reserved for system
  OB81_RESERVED_4 : BYTE ;	//Reserved for system
  OB81_RESERVED_5 : BYTE ;	//Reserved for system
  OB81_RESERVED_6 : BYTE ;	//Reserved for system
  OB81_DATE_TIME : DATE_AND_TIME ;	//Date and time OB81 started
END_VAR
BEGIN
// (block stored without names or comments; labels and parameter names are numbered)
END_ORGANIZATION_BLOCK

ORGANIZATION_BLOCK "HATAUYARISI"	// OB 82
TITLE = "I/O Point Fault"
VERSION : 0.1
VAR_TEMP
  OB82_EV_CLASS : BYTE ;	//16#39, Event class 3, Entering event state, Internal fault event
  OB82_FLT_ID : BYTE ;	//16#XX, Fault identifcation code
  OB82_PRIORITY : BYTE ;	//Priority of OB Execution
  OB82_OB_NUMBR : BYTE ;	//82 (Organization block 82, OB82)
  OB82_RESERVED_1 : BYTE ;	//Reserved for system
  OB82_IO_FLAG : BYTE ;	//Input (01010100), Output (01010101)
  OB82_MDL_ADDR : WORD ;	//Base address of module with fault
  OB82_MDL_DEFECT : BOOL ;	//Module defective
  OB82_INT_FAULT : BOOL ;	//Internal fault
  OB82_EXT_FAULT : BOOL ;	//External fault
  OB82_PNT_INFO : BOOL ;	//Point information
  OB82_EXT_VOLTAGE : BOOL ;	//External voltage low
  OB82_FLD_CONNCTR : BOOL ;	//Field wiring connector missing
  OB82_NO_CONFIG : BOOL ;	//Module has no configuration data
  OB82_CONFIG_ERR : BOOL ;	//Module has configuration error
  OB82_MDL_TYPE : BYTE ;	//Type of module
  OB82_SUB_MDL_ERR : BOOL ;	//Sub-Module is missing or has error
  OB82_COMM_FAULT : BOOL ;	//Communication fault
  OB82_MDL_STOP : BOOL ;	//Module is stopped
  OB82_WTCH_DOG_FLT : BOOL ;	//Watch dog timer stopped module
  OB82_INT_PS_FLT : BOOL ;	//Internal power supply fault
  OB82_PRIM_BATT_FLT : BOOL ;	//Primary battery is in fault
  OB82_BCKUP_BATT_FLT : BOOL ;	//Backup battery is in fault
  OB82_RESERVED_2 : BOOL ;	//Reserved for system
  OB82_RACK_FLT : BOOL ;	//Rack fault, only for bus interface module
  OB82_PROC_FLT : BOOL ;	//Processor fault
  OB82_EPROM_FLT : BOOL ;	//EPROM fault
  OB82_RAM_FLT : BOOL ;	//RAM fault
  OB82_ADU_FLT : BOOL ;	//ADU fault
  OB82_FUSE_FLT : BOOL ;	//Fuse fault
  OB82_HW_INTR_FLT : BOOL ;	//Hardware interupt input in fault
  OB82_RESERVED_3 : BOOL ;	//Reserved for system
  OB82_DATE_TIME : DATE_AND_TIME ;	//Date and time OB82 started
END_VAR
BEGIN
// (block stored without names or comments; labels and parameter names are numbered)
END_ORGANIZATION_BLOCK

ORGANIZATION_BLOCK "TAKMACIKARMAHATASI"	// OB 83
TITLE = "I/O Point Fault"
VERSION : 0.1
VAR_TEMP
  OB83_EV_CLASS : BYTE ;	//16#38/39, Event class 3, module inserted/removed (8/9)
  OB83_FLT_ID : BYTE ;	//16#XX, Fault identifcation code
  OB83_PRIORITY : BYTE ;	//Priority of OB Execution
  OB83_OB_NUMBR : BYTE ;	//83 (Organization block 83, OB83)
  OB83_RESERVED_1 : BYTE ;	//Reserved for system
  OB83_MDL_ID : BYTE ;	//Input module (01010100), Output module (01010101)
  OB83_MDL_ADDR : WORD ;	//Base address of module with point fault
  OB83_RACK_NUM : INT ;	//Number of rack that has module with point fault
  OB83_MDL_TYPE : WORD ;	//Module type with point fault
  OB83_DATE_TIME : DATE_AND_TIME ;	//Date and time OB83 started
END_VAR
BEGIN
// (block stored without names or comments; labels and parameter names are numbered)
END_ORGANIZATION_BLOCK

ORGANIZATION_BLOCK "CPUHARDWAREERROR"	// OB 84
TITLE = "CPU Fault"
VERSION : 0.1
VAR_TEMP
  OB84_EV_CLASS : BYTE ;	//16#38/39, Event class 3, module inserted/removed (8/9)
  OB84_FLT_ID : BYTE ;	//16#81, Fault identifcation code
  OB84_PRIORITY : BYTE ;	//Priority of OB Execution
  OB84_OB_NUMBR : BYTE ;	//84 (Organization block 84, OB84)
  OB84_RESERVED_1 : BYTE ;	//Reserved for system
  OB84_RESERVED_2 : BYTE ;	//Reserved for system
  OB84_RESERVED_3 : WORD ;	//Reserved for system
  OB84_RESERVED_4 : DWORD ;	//Reserved for system
  OB84_DATE_TIME : DATE_AND_TIME ;	//Date and time OB84 started
END_VAR
BEGIN
// (block stored without names or comments; labels and parameter names are numbered)
END_ORGANIZATION_BLOCK

ORGANIZATION_BLOCK "PROGRAMHATASI"	// OB 85
TITLE = "Organization Block (OB) Not Loaded Fault"
VERSION : 0.1
VAR_TEMP
  OB85_EV_CLASS : BYTE ;	//16#35 Event class 3
  OB85_FLT_ID : BYTE ;	//16#XX, Fault identification code
  OB85_PRIORITY : BYTE ;	//Priority of OB Execution
  OB85_OB_NUMBR : BYTE ;	//85 (Organization block 85, OB85)
  OB85_RESERVED_1 : BYTE ;	//Reserved for system
  OB85_RESERVED_2 : BYTE ;	//Reserved for system
  OB85_RESERVED_3 : INT ;	//Reserved for system
  OB85_ERR_EV_CLASS : BYTE ;	//Class of event causing error
  OB85_ERR_EV_NUM : BYTE ;	//Number of event causing error
  OB85_OB_PRIOR : BYTE ;	//Priority of OB causing error
  OB85_OB_NUM : BYTE ;	//Number of OB causing error
  OB85_DATE_TIME : DATE_AND_TIME ;	//Date and time OB85 started
END_VAR
BEGIN
// (block stored without names or comments; labels and parameter names are numbered)
END_ORGANIZATION_BLOCK

ORGANIZATION_BLOCK "RACKHATASI"	// OB 86
TITLE = "Loss Of Rack Fault"
VERSION : 0.1
VAR_TEMP
  OB86_EV_CLASS : BYTE ;	//16#38/39 Event class 3
  OB86_FLT_ID : BYTE ;	//16#C1/C4/C5, Fault identifcation code
  OB86_PRIORITY : BYTE ;	//Priority of OB Execution
  OB86_OB_NUMBR : BYTE ;	//86 (Organization block 86, OB86)
  OB86_RESERVED_1 : BYTE ;	//Reserved for system
  OB86_RESERVED_2 : BYTE ;	//Reserved for system
  OB86_MDL_ADDR : WORD ;	//Base address of IM module in rack with fault
  OB86_RACKS_FLTD : ARRAY  [0 .. 31 ] OF BOOL ;	//Racks in fault
  OB86_DATE_TIME : DATE_AND_TIME ;	//Date and time OB86 started
END_VAR
BEGIN
// (block stored without names or comments; labels and parameter names are numbered)
END_ORGANIZATION_BLOCK

ORGANIZATION_BLOCK "HABERLESMEHATASI"	// OB 87
TITLE = "Communication Fault"
VERSION : 0.1
VAR_TEMP
  OB87_EV_CLASS : BYTE ;	//16#39 Event class 3
  OB87_FLT_ID : BYTE ;	//16#XX, Fault identifcation code
  OB87_PRIORITY : BYTE ;	//Priority of OB Execution
  OB87_OB_NUMBR : BYTE ;	//87 (Organization block 87, OB87)
  OB87_RESERVED_1 : BYTE ;	//Reserved for system
  OB87_RESERVED_2 : BYTE ;	//Reserved for system
  OB87_RESERVED_3 : WORD ;	//Reserved for system
  OB87_RESERVED_4 : DWORD ;	//Reserved for system
  OB87_DATE_TIME : DATE_AND_TIME ;	//Date and time OB87 started
END_VAR
BEGIN
// (block stored without names or comments; labels and parameter names are numbered)
END_ORGANIZATION_BLOCK

ORGANIZATION_BLOCK "COMPLETE RESTART"	// OB 100
TITLE = "Complete Restart"
VERSION : 0.1
VAR_TEMP
  OB100_EV_CLASS : BYTE ;	//16#13, Event class 1, Entering event state, Event logged in diagnostic buffer
  OB100_STRTUP : BYTE ;	//16#81/82/83/84 Method of startup
  OB100_PRIORITY : BYTE ;	//Priority of OB Execution
  OB100_OB_NUMBR : BYTE ;	//100 (Organization block 100, OB100)
  OB100_RESERVED_1 : BYTE ;	//Reserved for system
  OB100_RESERVED_2 : BYTE ;	//Reserved for system
  OB100_STOP : WORD ;	//Event that caused CPU to stop (16#4xxx)
  OB100_STRT_INFO : DWORD ;	//Information on how system started
  OB100_DATE_TIME : DATE_AND_TIME ;	//Date and time OB100 started
END_VAR
BEGIN
NETWORK
TITLE = Kazan islemlerini sifirlama islemleri
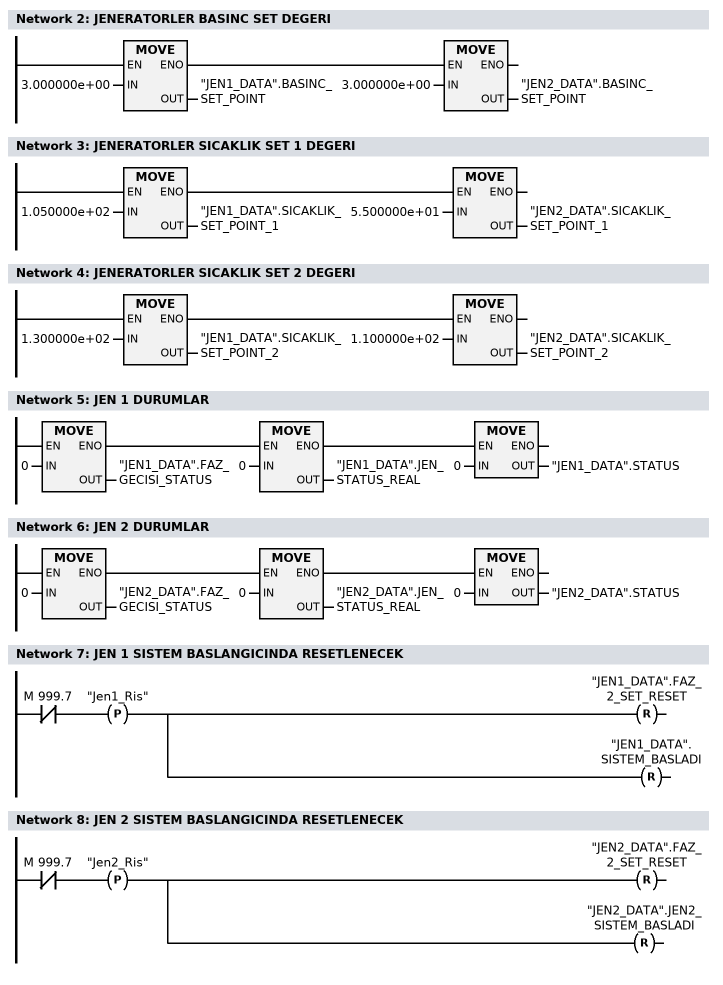
NETWORK
TITLE = JENERATORLER BASINC SET DEGERI
      A(;
      L     3.000000e+00;
      T     "JEN1_DATA".BASINC_SET_POINT;
      SET;
      SAVE;
      CLR;
      A     BR;
      );
      JNB   _001;
      L     3.000000e+00;
      T     "JEN2_DATA".BASINC_SET_POINT;
_001: NOP   0;
NETWORK
TITLE = JENERATORLER SICAKLIK SET 1 DEGERI
      A(;
      L     1.050000e+02;
      T     "JEN1_DATA".SICAKLIK_SET_POINT_1;
      SET;
      SAVE;
      CLR;
      A     BR;
      );
      JNB   _002;
      L     5.500000e+01;
      T     "JEN2_DATA".SICAKLIK_SET_POINT_1;
_002: NOP   0;
NETWORK
TITLE = JENERATORLER SICAKLIK SET 2 DEGERI
      A(;
      L     1.300000e+02;
      T     "JEN1_DATA".SICAKLIK_SET_POINT_2;
      SET;
      SAVE;
      CLR;
      A     BR;
      );
      JNB   _003;
      L     1.100000e+02;
      T     "JEN2_DATA".SICAKLIK_SET_POINT_2;
_003: NOP   0;
NETWORK
TITLE = JEN 1 DURUMLAR
      A(;
      A(;
      L     0;
      T     "JEN1_DATA".FAZ_GECISI_STATUS;
      SET;
      SAVE;
      CLR;
      A     BR;
      );
      JNB   _004;
      L     0;
      T     "JEN1_DATA".JEN_STATUS_REAL;
      SET;
      SAVE;
      CLR;
_004: A     BR;
      );
      JNB   _005;
      L     0;
      T     "JEN1_DATA".STATUS;
_005: NOP   0;
NETWORK
TITLE = JEN 2 DURUMLAR
      A(;
      A(;
      L     0;
      T     "JEN2_DATA".FAZ_GECISI_STATUS;
      SET;
      SAVE;
      CLR;
      A     BR;
      );
      JNB   _006;
      L     0;
      T     "JEN2_DATA".JEN_STATUS_REAL;
      SET;
      SAVE;
      CLR;
_006: A     BR;
      );
      JNB   _007;
      L     0;
      T     "JEN2_DATA".STATUS;
_007: NOP   0;
NETWORK
TITLE = JEN 1 SISTEM BASLANGICINDA RESETLENECEK
      AN    M 999.7;
      FP    "Jen1_Ris";
      R     "JEN1_DATA".FAZ_2_SET_RESET;
      R     "JEN1_DATA".SISTEM_BASLADI;
NETWORK
TITLE = JEN 2 SISTEM BASLANGICINDA RESETLENECEK
      AN    M 999.7;
      FP    "Jen2_Ris";
      R     "JEN2_DATA".FAZ_2_SET_RESET;
      R     "JEN2_DATA".JEN2_SISTEM_BASLADI;
END_ORGANIZATION_BLOCK

ORGANIZATION_BLOCK "RESTART"	// OB 101
TITLE = "Restart"
VERSION : 0.1
VAR_TEMP
  OB101_EV_CLASS : BYTE ;	//16#13, Event class 1, Entering event state, Event logged in diagnostic buffer
  OB101_STRTUP : BYTE ;	//16#81/82/83/84 Method of startup
  OB101_PRIORITY : BYTE ;	//Priority of OB Execution
  OB101_OB_NUMBR : BYTE ;	//101 (Organization block 101, OB101)
  OB101_RESERVED_1 : BYTE ;	//Reserved for system
  OB101_RESERVED_2 : BYTE ;	//Reserved for system
  OB101_STOP : WORD ;	//Event that caused CPU to stop (16#4xxx)
  OB101_STRT_INFO : DWORD ;	//Information on how system started
  OB101_DATE_TIME : DATE_AND_TIME ;	//Date and time OB101 started
END_VAR
BEGIN
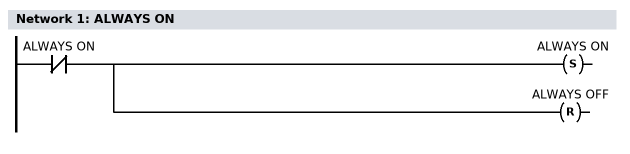
NETWORK
TITLE = ALWAYS ON
      AN    "ALWAYS ON";
      S     "ALWAYS ON";
      R     "ALWAYS OFF";
END_ORGANIZATION_BLOCK

ORGANIZATION_BLOCK "COLD RESTART"	// OB 102
TITLE = "Cold Restart"
VERSION : 0.1
VAR_TEMP
  OB102_EV_CLASS : BYTE ;	//16#13, Event class 1, Entering event state, Event logged in diagnostic buffer
  OB102_STRTUP : BYTE ;	//16#85...8B Method of startup
  OB102_PRIORITY : BYTE ;	//Priority of OB Execution
  OB102_OB_NUMBR : BYTE ;	//102 (Organization block 102, OB102)
  OB102_RESERVED_1 : BYTE ;	//Reserved for system
  OB102_RESERVED_2 : BYTE ;	//Reserved for system
  OB102_STOP : WORD ;	//Event that caused CPU to stop (16#4xxx)
  OB102_STRT_INFO : DWORD ;	//Information on how system started
  OB102_DATE_TIME : DATE_AND_TIME ;	//Date and time OB102 started
END_VAR
BEGIN
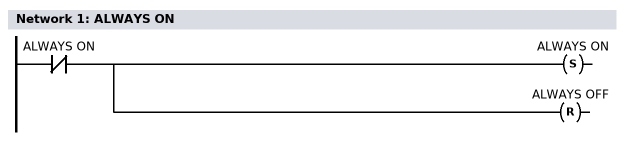
NETWORK
TITLE = ALWAYS ON
      AN    "ALWAYS ON";
      S     "ALWAYS ON";
      R     "ALWAYS OFF";
END_ORGANIZATION_BLOCK

ORGANIZATION_BLOCK "PROGRAMMINGERROR"	// OB 121
TITLE = "Programming Error"
VERSION : 0.1
VAR_TEMP
  OB121_EV_CLASS : BYTE ;	//16#25, Event class 2, Entering event state, Internal fault event
  OB121_SW_FLT : BYTE ;	//16#XX Software programming fault
  OB121_PRIORITY : BYTE ;	//Priority of OB Execution
  OB121_OB_NUMBR : BYTE ;	//121 (Organization block 121, OB121)
  OB121_BLK_TYPE : BYTE ;	//16#88/8A/8B/8C/8E Type of block fault occured in
  OB121_RESERVED_1 : BYTE ;	//Reserved for system
  OB121_FLT_REG : WORD ;	//16#XX Specific register that caused fault
  OB121_BLK_NUM : WORD ;	//Number of block that programming fault occured in
  OB121_PRG_ADDR : WORD ;	//Address in block where programming fault occured
  OB121_DATE_TIME : DATE_AND_TIME ;	//Date and time OB121 started
END_VAR
BEGIN
// (block stored without names or comments; labels and parameter names are numbered)
END_ORGANIZATION_BLOCK

ORGANIZATION_BLOCK "MOD_ERR"	// OB 122
TITLE = "Module Access Error"
VERSION : 0.1
VAR_TEMP
  OB122_EV_CLASS : BYTE ;	//16#29, Event class 2, Entering event state, Internal fault event
  OB122_SW_FLT : BYTE ;	//16#XX Software error code
  OB122_PRIORITY : BYTE ;	//Priority of OB Execution
  OB122_OB_NUMBR : BYTE ;	//122 (Organization block 122, OB122)
  OB122_BLK_TYPE : BYTE ;	//16#88/8C/8E Type of block fault occured in
  OB122_MEM_AREA : BYTE ;	//Memory area where access error occured
  OB122_MEM_ADDR : WORD ;	//Memory address where access error occured
  OB122_BLK_NUM : WORD ;	//Block number in which error occured
  OB122_PRG_ADDR : WORD ;	//Program address where error occured
  OB122_DATE_TIME : DATE_AND_TIME ;	//Date and time OB1 started
END_VAR
BEGIN
// (block stored without names or comments; labels and parameter names are numbered)
END_ORGANIZATION_BLOCK

// (several symbol tables fit these blocks; global names not applied)

FUNCTION_BLOCK FB 1
VERSION : 0.1
BEGIN
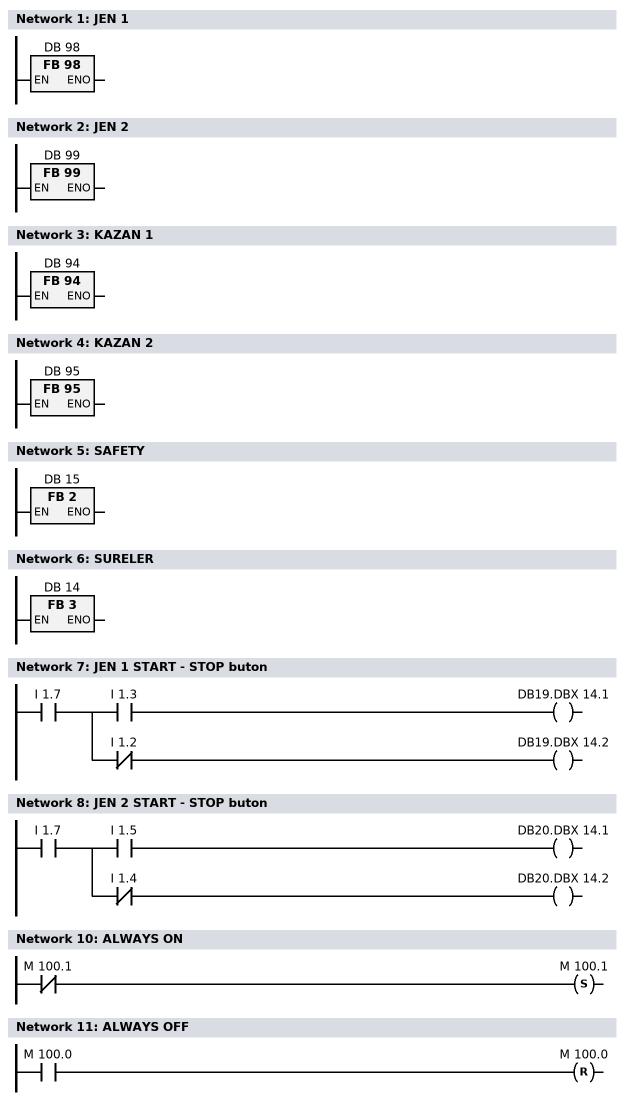
NETWORK
TITLE = JEN 1
      CALL  FB 98 , DB 98;
      NOP   0;
NETWORK
TITLE = JEN 2
      CALL  FB 99 , DB 99;
      NOP   0;
NETWORK
TITLE = KAZAN 1
      CALL  FB 94 , DB 94;
      NOP   0;
NETWORK
TITLE = KAZAN 2
      CALL  FB 95 , DB 95;
      NOP   0;
NETWORK
TITLE = SAFETY
      CALL  FB 2 , DB 15;
      NOP   0;
NETWORK
TITLE = SURELER
      CALL  FB 3 , DB 14;
      NOP   0;
NETWORK
TITLE = JEN 1 START - STOP buton
      A     I 1.7;
      =     L 0.0;
      A     L 0.0;
      A     I 1.3;
      =     DB19.DBX 14.1;
      A     L 0.0;
      AN    I 1.2;
      =     DB19.DBX 14.2;
NETWORK
TITLE = JEN 2 START - STOP buton
      A     I 1.7;
      =     L 0.0;
      A     L 0.0;
      A     I 1.5;
      =     DB20.DBX 14.1;
      A     L 0.0;
      AN    I 1.4;
      =     DB20.DBX 14.2;
NETWORK
TITLE =
NETWORK
TITLE = ALWAYS ON
      AN    M 100.1;
      S     M 100.1;
NETWORK
TITLE = ALWAYS OFF
      A     M 100.0;
      R     M 100.0;
NETWORK
TITLE =
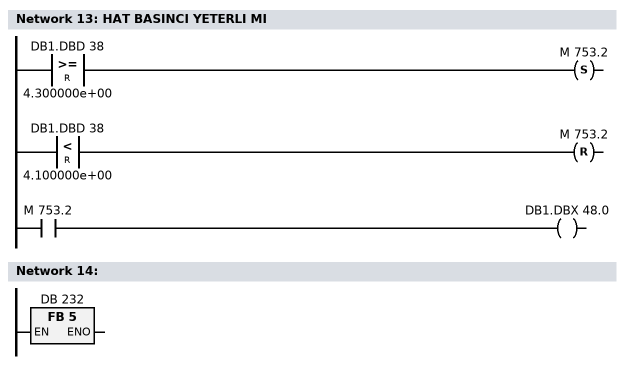
NETWORK
TITLE = HAT BASINCI YETERLI MI
      A(;
      L     DB1.DBD 38;
      L     4.300000e+00;
      >=R;
      );
      S     M 753.2;
      A(;
      L     DB1.DBD 38;
      L     4.100000e+00;
      <R;
      );
      R     M 753.2;
      A     M 753.2;
      =     DB1.DBX 48.0;
NETWORK
TITLE =
      CALL  FB 5 , DB 232;
      NOP   0;
END_FUNCTION_BLOCK

FUNCTION_BLOCK FB 2
VERSION : 0.1
BEGIN
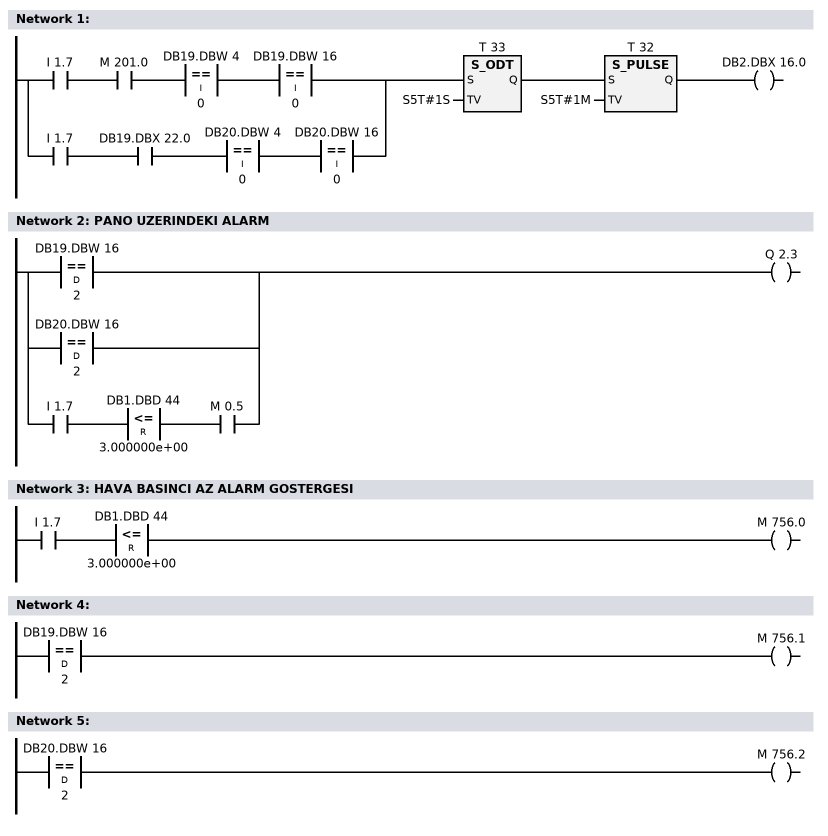
NETWORK
TITLE =
      A(;
      A(;
      A     I 1.7;
      A     M 201.0;
      A(;
      L     DB19.DBW 4;
      L     0;
      ==I;
      );
      A(;
      L     DB19.DBW 16;
      L     0;
      ==I;
      );
      O;
      A     I 1.7;
      A     DB19.DBX 22.0;
      A(;
      L     DB20.DBW 4;
      L     0;
      ==I;
      );
      A(;
      L     DB20.DBW 16;
      L     0;
      ==I;
      );
      );
      L     S5T#1S;
      SD    T 33;
      NOP   0;
      NOP   0;
      NOP   0;
      A     T 33;
      );
      L     S5T#1M;
      SP    T 32;
      NOP   0;
      NOP   0;
      NOP   0;
      A     T 32;
      =     DB2.DBX 16.0;
NETWORK
TITLE = PANO UZERINDEKI ALARM 
//JENERATORDE MINIMUM SU SEVIYESINE DUSERSE PANO UZERINDEKI ALARMI CALISTIR
      O(;
      L     DB19.DBW 16;
      L     2;
      ==D;
      );
      O(;
      L     DB20.DBW 16;
      L     2;
      ==D;
      );
      O;
      A     I 1.7;
      A(;
      L     DB1.DBD 44;
      L     3.000000e+00;
      <=R;
      );
      A     M 0.5;
      =     Q 2.3;
NETWORK
TITLE = HAVA BASINCI AZ ALARM GOSTERGESI
      A     I 1.7;
      A(;
      L     DB1.DBD 44;
      L     3.000000e+00;
      <=R;
      );
      =     M 756.0;
NETWORK
TITLE =
      L     DB19.DBW 16;
      L     2;
      ==D;
      =     M 756.1;
NETWORK
TITLE =
      L     DB20.DBW 16;
      L     2;
      ==D;
      =     M 756.2;
END_FUNCTION_BLOCK

FUNCTION_BLOCK FB 3
VERSION : 0.1
BEGIN
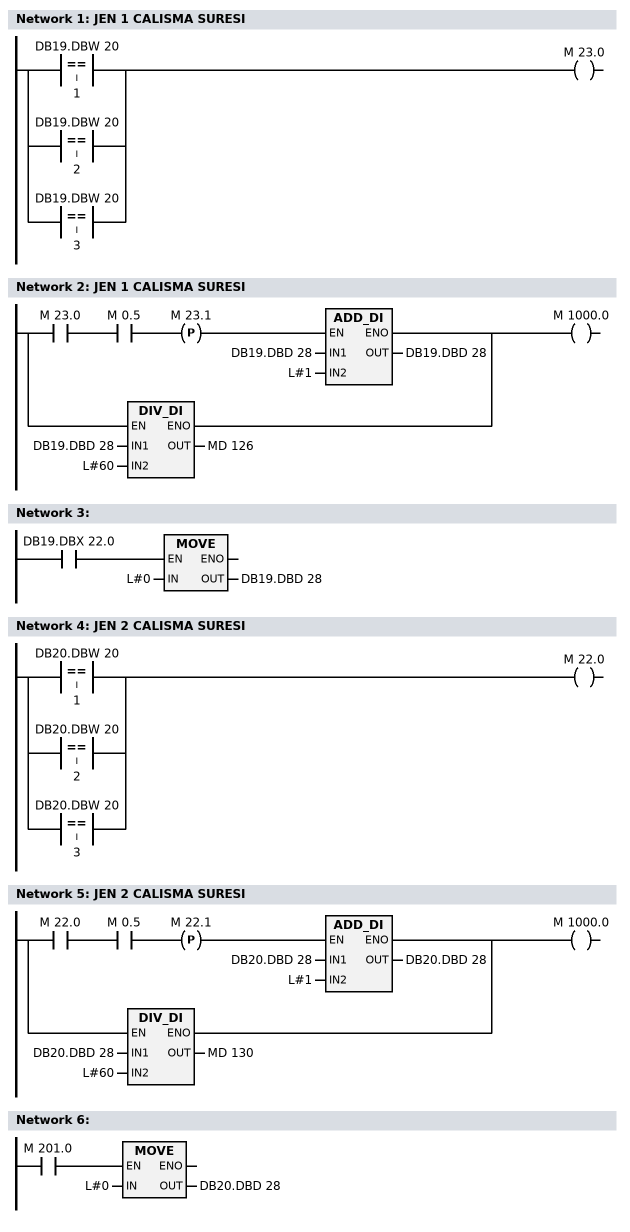
NETWORK
TITLE = JEN 1 CALISMA SURESI
      O(;
      L     DB19.DBW 20;
      L     1;
      ==I;
      );
      O(;
      L     DB19.DBW 20;
      L     2;
      ==I;
      );
      O(;
      L     DB19.DBW 20;
      L     3;
      ==I;
      );
      =     M 23.0;
NETWORK
TITLE = JEN 1 CALISMA SURESI
      O(;
      A     M 23.0;
      A     M 0.5;
      FP    M 23.1;
      JNB   _001;
      L     DB19.DBD 28;
      L     L#1;
      +D;
      T     DB19.DBD 28;
      AN    OV;
      SAVE;
      CLR;
_001: A     BR;
      );
      O(;
      L     DB19.DBD 28;
      L     L#60;
      /D;
      T     MD 126;
      AN    OV;
      SAVE;
      CLR;
      A     BR;
      );
      =     M 1000.0;
NETWORK
TITLE =
      A     DB19.DBX 22.0;
      JNB   _002;
      L     L#0;
      T     DB19.DBD 28;
_002: NOP   0;
NETWORK
TITLE = JEN 2 CALISMA SURESI
      O(;
      L     DB20.DBW 20;
      L     1;
      ==I;
      );
      O(;
      L     DB20.DBW 20;
      L     2;
      ==I;
      );
      O(;
      L     DB20.DBW 20;
      L     3;
      ==I;
      );
      =     M 22.0;
NETWORK
TITLE = JEN 2 CALISMA SURESI
      O(;
      A     M 22.0;
      A     M 0.5;
      FP    M 22.1;
      JNB   _003;
      L     DB20.DBD 28;
      L     L#1;
      +D;
      T     DB20.DBD 28;
      AN    OV;
      SAVE;
      CLR;
_003: A     BR;
      );
      O(;
      L     DB20.DBD 28;
      L     L#60;
      /D;
      T     MD 130;
      AN    OV;
      SAVE;
      CLR;
      A     BR;
      );
      =     M 1000.0;
NETWORK
TITLE =
      A     M 201.0;
      JNB   _004;
      L     L#0;
      T     DB20.DBD 28;
_004: NOP   0;
NETWORK
TITLE = OTOKLAV 1 PISIM GECEN SURE
      O(;
      A(;
      A     DB17.DBX 40.3;
      =     L 0.0;
      BLD   103;
      BLD   9;
      =     L 5.0;
      CDB;
      OPN   DI 5;
      TAR2  LD 1;
      A     L 0.0;
      =     DIX 0.0;
      L     L#82800000;
      T     DID 2;
      LAR2  P#DBX 0.0;
      UC    SFB 4;
      LAR2  LD 1;
      L     DID 8;
      OPN   DI 17;
      T     DID 42;
      OPN   DI 5;
      CDB;
      BLD   10;
      A     BR;
      );
      JNB   _005;
      CALL  FC 1 (
           iTimeET                  := DB17.DBD 42,
           iIstenileSure            := DB17.DBW 4,
           oOUT                     := DB17.DBD 46);
_005: A     BR;
      );
      O(;
      L     DB17.DBD 46;
      L     60;
      /D;
      T     MD 118;
      AN    OV;
      SAVE;
      CLR;
      A     BR;
      );
      =     M 1000.0;
NETWORK
TITLE = OTOKLAV 2 PISIM GECEN SURE
      O(;
      A(;
      A     DB18.DBX 40.3;
      =     L 0.0;
      BLD   103;
      BLD   9;
      =     L 5.0;
      CDB;
      OPN   DI 6;
      TAR2  LD 1;
      A     L 0.0;
      =     DIX 0.0;
      L     L#82800000;
      T     DID 2;
      LAR2  P#DBX 0.0;
      UC    SFB 4;
      LAR2  LD 1;
      L     DID 8;
      OPN   DI 18;
      T     DID 42;
      OPN   DI 6;
      CDB;
      BLD   10;
      A     BR;
      );
      JNB   _006;
      CALL  FC 1 (
           iTimeET                  := DB18.DBD 42,
           iIstenileSure            := DB18.DBW 4,
           oOUT                     := DB18.DBD 46);
_006: A     BR;
      );
      O(;
      L     DB18.DBD 46;
      L     60;
      /D;
      T     MD 122;
      AN    OV;
      SAVE;
      CLR;
      A     BR;
      );
      =     M 1000.0;
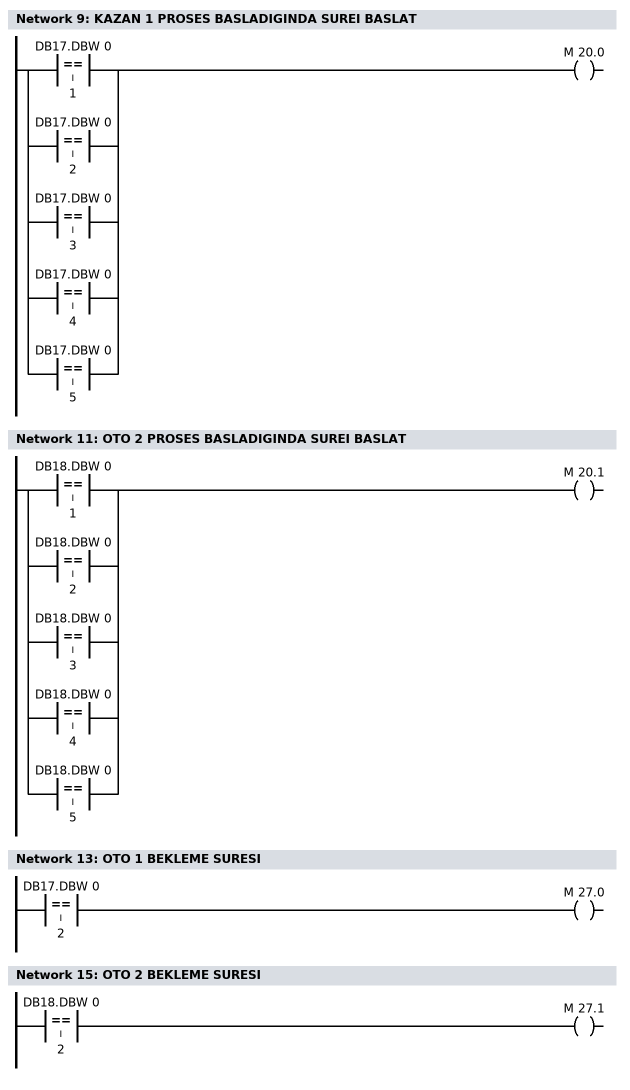
NETWORK
TITLE = KAZAN 1 PROSES BASLADIGINDA SUREI BASLAT
      O(;
      L     DB17.DBW 0;
      L     1;
      ==I;
      );
      O(;
      L     DB17.DBW 0;
      L     2;
      ==I;
      );
      O(;
      L     DB17.DBW 0;
      L     3;
      ==I;
      );
      O(;
      L     DB17.DBW 0;
      L     4;
      ==I;
      );
      O(;
      L     DB17.DBW 0;
      L     5;
      ==I;
      );
      =     M 20.0;
NETWORK
TITLE = OTOKLAV 1 PROSES SURESI
      O(;
      A(;
      A     M 20.0;
      =     L 0.0;
      BLD   103;
      BLD   9;
      =     L 5.0;
      CDB;
      OPN   DI 7;
      TAR2  LD 1;
      A     L 0.0;
      =     DIX 0.0;
      L     L#82800000;
      T     DID 2;
      LAR2  P#DBX 0.0;
      UC    SFB 4;
      LAR2  LD 1;
      L     DID 8;
      OPN   DI 17;
      T     DID 50;
      OPN   DI 7;
      CDB;
      BLD   10;
      A     BR;
      );
      JNB   _007;
      L     DB17.DBD 50;
      L     1000;
      /D;
      T     DB17.DBD 54;
      AN    OV;
      SAVE;
      CLR;
_007: A     BR;
      );
      O(;
      L     DB17.DBD 54;
      L     60;
      /D;
      T     MD 110;
      AN    OV;
      SAVE;
      CLR;
      A     BR;
      );
      =     M 1000.0;
NETWORK
TITLE = OTO 2 PROSES BASLADIGINDA SUREI BASLAT
      O(;
      L     DB18.DBW 0;
      L     1;
      ==I;
      );
      O(;
      L     DB18.DBW 0;
      L     2;
      ==I;
      );
      O(;
      L     DB18.DBW 0;
      L     3;
      ==I;
      );
      O(;
      L     DB18.DBW 0;
      L     4;
      ==I;
      );
      O(;
      L     DB18.DBW 0;
      L     5;
      ==I;
      );
      =     M 20.1;
NETWORK
TITLE = OTO 2 PROSES_SURESI
      O(;
      A(;
      A     M 20.1;
      =     L 0.0;
      BLD   103;
      BLD   9;
      =     L 5.0;
      CDB;
      OPN   DI 8;
      TAR2  LD 1;
      A     L 0.0;
      =     DIX 0.0;
      L     L#82800000;
      T     DID 2;
      LAR2  P#DBX 0.0;
      UC    SFB 4;
      LAR2  LD 1;
      L     DID 8;
      OPN   DI 18;
      T     DID 50;
      OPN   DI 8;
      CDB;
      BLD   10;
      A     BR;
      );
      JNB   _008;
      L     DB18.DBD 50;
      L     1000;
      /D;
      T     DB18.DBD 54;
      AN    OV;
      SAVE;
      CLR;
_008: A     BR;
      );
      O(;
      L     DB18.DBD 54;
      L     60;
      /D;
      T     MD 114;
      AN    OV;
      SAVE;
      CLR;
      A     BR;
      );
      =     M 1000.0;
NETWORK
TITLE = OTO 1 BEKLEME SURESI
      L     DB17.DBW 0;
      L     2;
      ==I;
      =     M 27.0;
NETWORK
TITLE = OTO 1 BEKLEME SURESI
      A(;
      A     M 27.0;
      =     L 0.0;
      BLD   103;
      BLD   9;
      =     L 5.0;
      CDB;
      OPN   DI 9;
      TAR2  LD 1;
      A     L 0.0;
      =     DIX 0.0;
      L     L#82800000;
      T     DID 2;
      LAR2  P#DBX 0.0;
      UC    SFB 4;
      LAR2  LD 1;
      L     DID 8;
      OPN   DI 17;
      T     DID 58;
      OPN   DI 9;
      CDB;
      BLD   10;
      A     BR;
      );
      JNB   _009;
      L     DB17.DBD 58;
      L     1000;
      /D;
      T     DB17.DBD 62;
_009: NOP   0;
NETWORK
TITLE = OTO 2 BEKLEME SURESI
      L     DB18.DBW 0;
      L     2;
      ==I;
      =     M 27.1;
NETWORK
TITLE = OTO 2 BEKLEME SURESI
      A(;
      A     M 27.1;
      =     L 0.0;
      BLD   103;
      BLD   9;
      =     L 5.0;
      CDB;
      OPN   DI 10;
      TAR2  LD 1;
      A     L 0.0;
      =     DIX 0.0;
      L     L#82800000;
      T     DID 2;
      LAR2  P#DBX 0.0;
      UC    SFB 4;
      LAR2  LD 1;
      L     DID 8;
      OPN   DI 18;
      T     DID 58;
      OPN   DI 10;
      CDB;
      BLD   10;
      A     BR;
      );
      JNB   _00a;
      L     DB18.DBD 58;
      L     1000;
      /D;
      T     DB18.DBD 62;
_00a: NOP   0;
END_FUNCTION_BLOCK

FUNCTION_BLOCK FB 5
VERSION : 0.1
BEGIN
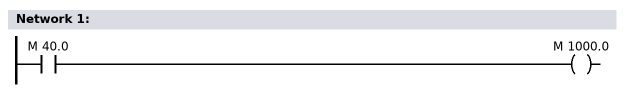
NETWORK
TITLE =
      A     M 40.0;
      =     M 1000.0;
END_FUNCTION_BLOCK

FUNCTION_BLOCK FB 20
//0 - baslama kriterleri
//1 - pid baslasin
//
VERSION : 0.1
VAR_INPUT
  IN_ACIL_STOP : BOOL ;
  IN_START : BOOL ;
  IN_TRANSFER : BOOL ;
  IN_BOSALTIM : BOOL ;
  IN_KAPAK : BOOL ;
  IN_JEN1_OK : BOOL ;
  IN_JEN2_OK : BOOL ;
  IN_JENS_OK : BOOL ;
  IN_TRANSFERE_HAZIR : BOOL ;
  IN_PISIM_SURESI : S5TIME ;
  IN_SCALE_BASINC_PER : INT ;
  IN_SET_BASINC : REAL ;
  IN_DIGER_KAZAN_BASINCI : REAL ;
  IN_TIMER_500MS : TIMER ;
  IN_TIMER_1S : TIMER ;
  IN_TIMER_PISIRME : TIMER ;
  IN_TIMER_500MS_2 : TIMER ;
  IN_TIMER_7S : TIMER ;
  IN_SCALE_HI_LIM : REAL ;
  IN_SCALE_LO_LIM : REAL ;
  IN_SCALE_SICAKLIK_HI_LIM : REAL ;
  IN_SCALE_SICAKLIK_LO_LIM : REAL ;
  IN_SCALE_SICAKLIK_PER : INT ;
  IN_DIGER_KAZAN_BOSALTIMD : BOOL ;
  IN_TRANSFER_BASLADI : BOOL ;
  IN_PISIM_SURESI_TIME_DB : BLOCK_DB ;
  IN_DIG_KAZAN_PROSES_BAS : BOOL ;
  IN_JEN_DURDU : BOOL ;
  IN_JEN_DURDUR_PID_MAN : REAL ;
  IN_DELAY_BITISI_BEKLE : TIMER ;
  IN_DELAY_BIRAZ_BEKLE : TIMER ;
END_VAR
VAR_OUTPUT
  O_YESIL_LAM : BOOL ;
  O_KIRMIZI_LAM : BOOL ;
  O_DUDUK : BOOL ;
  O_BOSALTIM_VALFI : BOOL ;
  O_PID_MAN_ON : BOOL ;
  O_PID_MAN : REAL ;
  O_TRANSFER_YAPILIYOR : BOOL ;
  O_SCALE_BASINC_RET_VAL : WORD ;
  O_SCALE_BASINC_OUT : REAL ;
  O_EMNIYET_VALFI : BOOL ;
  O_TRANSFERE_HAZIR : BOOL ;
  O_SCALE_SICAKLIK_RET_VAL : WORD ;
  O_SCALE_SICAKLIK_OUT : REAL ;
  O_TRANSFER_ET_LAMBASI : BOOL ;
  O_PROSES_BASLADI : BOOL ;
  O_KAZAN_BOSALTIMDA : BOOL ;
  O_PISIM_BASLADI : BOOL ;
END_VAR
VAR_IN_OUT
  STATUS : INT ;
END_VAR
VAR
  ST_STATUS : INT ;
  ST_OUT_BOSALTIM_MEM : BOOL ;
  ST_OUT_PID_MAN_ON : BOOL ;
  ST_OUT_PID_MAN : REAL ;
  st_ris_pid_zero : BOOL ;
  st_scale_hi_lim : REAL  := 1.000000e+001;
  st_scale_lo_lim : REAL ;
  st_basinc_ok_sure_basla : BOOL ;
  st_tolerans_mul : REAL ;
  st_toleransli_basinc : REAL ;
  st_adim4_bosaltim_valfi : BOOL ;
  st_OUT_adim4_emnyet_val : BOOL ;
  st_pid_basla : BOOL ;
  st_bosalti_valfi_acil : BOOL ;
  st_scale_basinc_ret_val : WORD ;
  st_scale_basinc_out : REAL ;
  st_scale_sicaklik_ret_va : WORD ;
  st_scale_sicaklik_out : REAL ;
  ST_PROSES_BASLADI : BOOL ;
  ST_KAZAN_BOSALTIMDA : BOOL ;
  ST_BOS : BOOL ;
  ST_SET_ADD_BASINC_02 : REAL ;
  ST_GECEN_PISIM_SURESI : TIME ;
  st_5_bar_ustu : BOOL ;
  st_5_bar_alti : BOOL ;
  st_5_bar_guvenlik_SR : BOOL ;
  st_5_bar_guvenlik_mem : BOOL ;
END_VAR
BEGIN
NETWORK
TITLE = BASLANGIC SARTLARI
      A(;
      A(;
      A     M 100.0;
      =     L 0.0;
      BLD   103;
      CALL  FC 105 (
           $1                       := #IN_SCALE_BASINC_PER,
           $2                       := #IN_SCALE_HI_LIM,
           $3                       := #IN_SCALE_LO_LIM,
           $4                       := L 0.0,
           $5                       := #st_scale_basinc_ret_val,
           $6                       := #st_scale_basinc_out);
      A     BR;
      );
      JNB   _001;
      L     #st_scale_basinc_ret_val;
      T     #O_SCALE_BASINC_RET_VAL;
      SET;
      SAVE;
      CLR;
_001: A     BR;
      );
      JNB   _002;
      L     #st_scale_basinc_out;
      T     #O_SCALE_BASINC_OUT;
_002: NOP   0;
NETWORK
TITLE =
      A(;
      A(;
      A     M 100.0;
      =     L 0.0;
      BLD   103;
      CALL  FC 105 (
           $1                       := #IN_SCALE_SICAKLIK_PER,
           $2                       := #IN_SCALE_SICAKLIK_HI_LIM,
           $3                       := #IN_SCALE_SICAKLIK_LO_LIM,
           $4                       := L 0.0,
           $5                       := #st_scale_sicaklik_ret_va,
           $6                       := #st_scale_sicaklik_out);
      A     BR;
      );
      JNB   _003;
      L     #st_scale_sicaklik_ret_va;
      T     #O_SCALE_SICAKLIK_RET_VAL;
      SET;
      SAVE;
      CLR;
_003: A     BR;
      );
      JNB   _004;
      L     #st_scale_sicaklik_out;
      T     #O_SCALE_SICAKLIK_OUT;
_004: NOP   0;
NETWORK
TITLE = START
      A(;
      A     I 1.7;
      A     #IN_ACIL_STOP;
      A     DB1.DBX 48.0;
      L     S5T#200MS;
      T     LD 0;
      TAK;
      T     LD 4;
      L     #IN_TIMER_500MS;
      T     LW 8;
      L     LD 4;
      L     LD 0;
      SD    T [LW 8];
      NOP   0;
      NOP   0;
      NOP   0;
      T     LD 0;
      TAK;
      T     LD 4;
      L     #IN_TIMER_500MS;
      T     LW 8;
      L     LD 4;
      L     LD 0;
      A     T [LW 8];
      );
      A     #IN_KAPAK;
      A     #IN_START;
      A(;
      L     #STATUS;
      L     0;
      ==I;
      );
      JNB   _005;
      L     1;
      T     #STATUS;
      SET;
      SAVE;
      CLR;
_005: A     BR;
      S     #ST_PROSES_BASLADI;
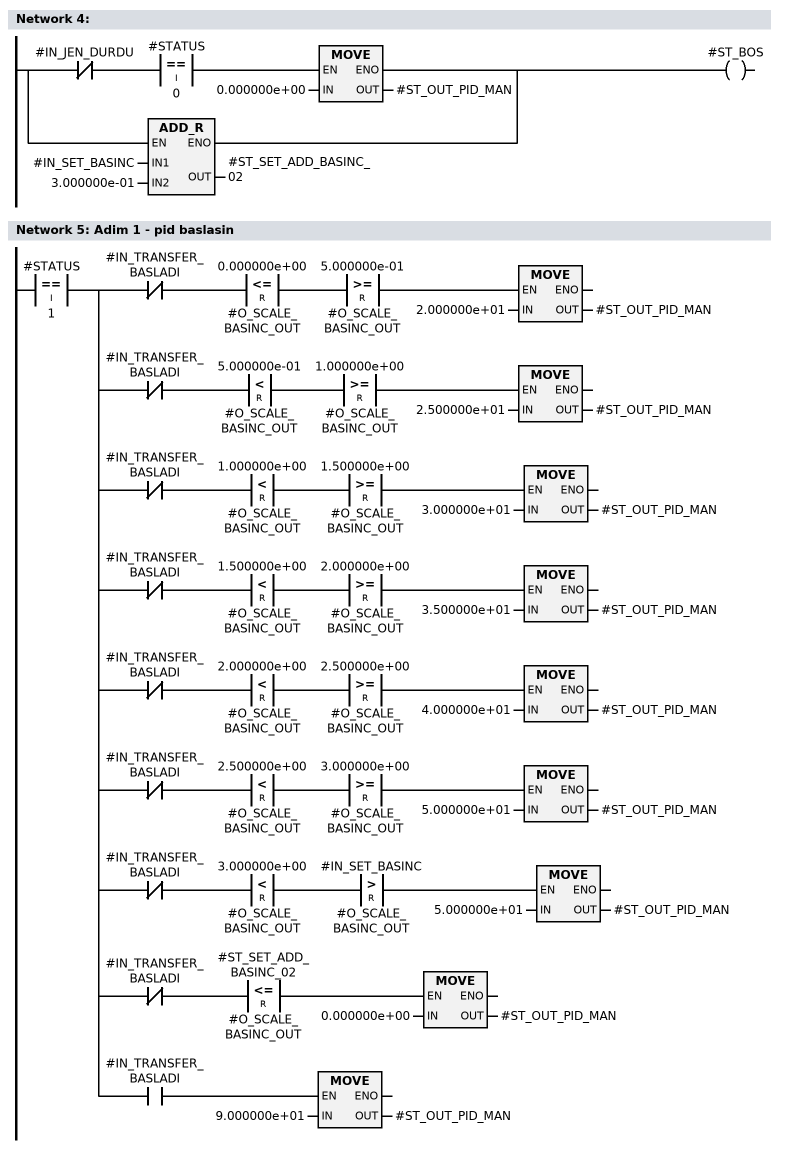
NETWORK
TITLE =
//1-Baslangicta vakum olmamasi icin bosaltim valfini ac
//Valf Normalde acik gibi dusundum
//2-Oransal valfi kapali tut
      O(;
      AN    #IN_JEN_DURDU;
      A(;
      L     #STATUS;
      L     0;
      ==I;
      );
      JNB   _006;
      L     0.000000e+00;
      T     #ST_OUT_PID_MAN;
      SET;
      SAVE;
      CLR;
_006: A     BR;
      );
      O(;
      L     #IN_SET_BASINC;
      L     3.000000e-01;
      +R;
      T     #ST_SET_ADD_BASINC_02;
      AN    OV;
      SAVE;
      CLR;
      A     BR;
      );
      =     #ST_BOS;
NETWORK
TITLE = Adim 1 - pid baslasin
      L     #STATUS;
      L     1;
      ==I;
      =     L 0.0;
      A     L 0.0;
      AN    #IN_TRANSFER_BASLADI;
      A(;
      L     0.000000e+00;
      L     #O_SCALE_BASINC_OUT;
      <=R;
      );
      A(;
      L     5.000000e-01;
      L     #O_SCALE_BASINC_OUT;
      >=R;
      );
      JNB   _007;
      L     2.000000e+01;
      T     #ST_OUT_PID_MAN;
_007: NOP   0;
      A     L 0.0;
      AN    #IN_TRANSFER_BASLADI;
      A(;
      L     5.000000e-01;
      L     #O_SCALE_BASINC_OUT;
      <R;
      );
      A(;
      L     1.000000e+00;
      L     #O_SCALE_BASINC_OUT;
      >=R;
      );
      JNB   _008;
      L     2.500000e+01;
      T     #ST_OUT_PID_MAN;
_008: NOP   0;
      A     L 0.0;
      AN    #IN_TRANSFER_BASLADI;
      A(;
      L     1.000000e+00;
      L     #O_SCALE_BASINC_OUT;
      <R;
      );
      A(;
      L     1.500000e+00;
      L     #O_SCALE_BASINC_OUT;
      >=R;
      );
      JNB   _009;
      L     3.000000e+01;
      T     #ST_OUT_PID_MAN;
_009: NOP   0;
      A     L 0.0;
      AN    #IN_TRANSFER_BASLADI;
      A(;
      L     1.500000e+00;
      L     #O_SCALE_BASINC_OUT;
      <R;
      );
      A(;
      L     2.000000e+00;
      L     #O_SCALE_BASINC_OUT;
      >=R;
      );
      JNB   _00a;
      L     3.500000e+01;
      T     #ST_OUT_PID_MAN;
_00a: NOP   0;
      A     L 0.0;
      AN    #IN_TRANSFER_BASLADI;
      A(;
      L     2.000000e+00;
      L     #O_SCALE_BASINC_OUT;
      <R;
      );
      A(;
      L     2.500000e+00;
      L     #O_SCALE_BASINC_OUT;
      >=R;
      );
      JNB   _00b;
      L     4.000000e+01;
      T     #ST_OUT_PID_MAN;
_00b: NOP   0;
      A     L 0.0;
      AN    #IN_TRANSFER_BASLADI;
      A(;
      L     2.500000e+00;
      L     #O_SCALE_BASINC_OUT;
      <R;
      );
      A(;
      L     3.000000e+00;
      L     #O_SCALE_BASINC_OUT;
      >=R;
      );
      JNB   _00c;
      L     5.000000e+01;
      T     #ST_OUT_PID_MAN;
_00c: NOP   0;
      A     L 0.0;
      AN    #IN_TRANSFER_BASLADI;
      A(;
      L     3.000000e+00;
      L     #O_SCALE_BASINC_OUT;
      <R;
      );
      A(;
      L     #IN_SET_BASINC;
      L     #O_SCALE_BASINC_OUT;
      >R;
      );
      JNB   _00d;
      L     5.000000e+01;
      T     #ST_OUT_PID_MAN;
_00d: NOP   0;
      A     L 0.0;
      AN    #IN_TRANSFER_BASLADI;
      A(;
      L     #ST_SET_ADD_BASINC_02;
      L     #O_SCALE_BASINC_OUT;
      <=R;
      );
      JNB   _00e;
      L     0.000000e+00;
      T     #ST_OUT_PID_MAN;
_00e: NOP   0;
      A     L 0.0;
      A     #IN_TRANSFER_BASLADI;
      JNB   _00f;
      L     9.000000e+01;
      T     #ST_OUT_PID_MAN;
_00f: NOP   0;
NETWORK
TITLE = Adim 1 - Pisim Süresi
      L     #STATUS;
      L     1;
      ==I;
      =     L 0.0;
      A(;
      A     L 0.0;
      A     #st_basinc_ok_sure_basla;
      L     #IN_PISIM_SURESI;
      T     LD 1;
      TAK;
      T     LD 5;
      L     #IN_TIMER_PISIRME;
      T     LW 9;
      L     LD 5;
      L     LD 1;
      SD    T [LW 9];
      NOP   0;
      NOP   0;
      NOP   0;
      T     LD 1;
      TAK;
      T     LD 5;
      L     #IN_TIMER_PISIRME;
      T     LW 9;
      L     LD 5;
      L     LD 1;
      A     T [LW 9];
      );
      JNB   _010;
      L     2;
      T     #STATUS;
_010: NOP   0;
      A     L 0.0;
      A(;
      O(;
      L     #O_SCALE_BASINC_OUT;
      L     #IN_SET_BASINC;
      >=R;
      );
      O     #st_basinc_ok_sure_basla;
      );
      =     #st_basinc_ok_sure_basla;
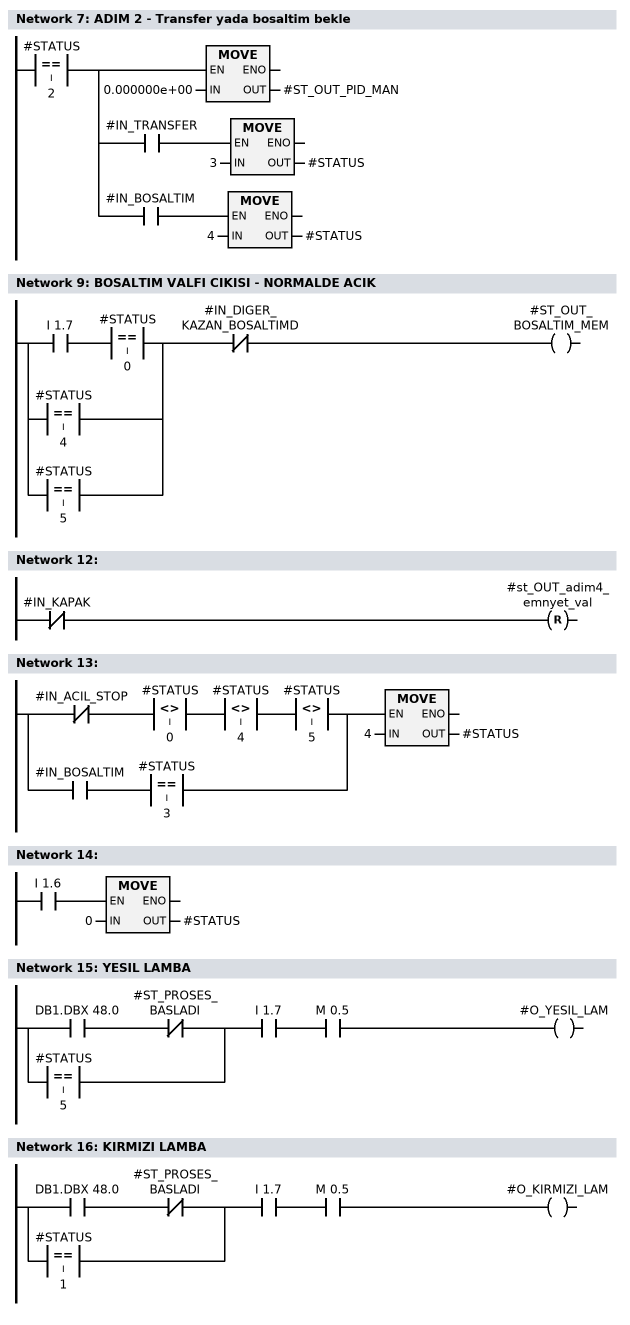
NETWORK
TITLE = ADIM 2 - Transfer yada bosaltim bekle
//1- Adim 2 Transfer ya da bosaltim bekle
//2- Oransal Vanayi kapali tut
      L     #STATUS;
      L     2;
      ==I;
      =     L 0.0;
      A     L 0.0;
      JNB   _011;
      L     0.000000e+00;
      T     #ST_OUT_PID_MAN;
_011: NOP   0;
      A     L 0.0;
      A     #IN_TRANSFER;
      JNB   _012;
      L     3;
      T     #STATUS;
_012: NOP   0;
      A     L 0.0;
      A     #IN_BOSALTIM;
      JNB   _013;
      L     4;
      T     #STATUS;
_013: NOP   0;
NETWORK
TITLE = Adim 3 - Transfer islemi
//1- Diger kazan hazir oldugunda transfer islmeini baslat
      A(;
      L     #STATUS;
      L     3;
      ==I;
      );
      A     #IN_TRANSFERE_HAZIR;
      JNB   _014;
      L     9.000000e+01;
      T     #ST_OUT_PID_MAN;
      SET;
      SAVE;
      CLR;
_014: A     BR;
      =     L 0.0;
      A     L 0.0;
      BLD   102;
      =     #O_TRANSFER_YAPILIYOR;
      A(;
      A     L 0.0;
      L     S5T#23S;
      T     LD 1;
      TAK;
      T     LD 5;
      L     #IN_TIMER_500MS_2;
      T     LW 9;
      L     LD 5;
      L     LD 1;
      SD    T [LW 9];
      NOP   0;
      NOP   0;
      NOP   0;
      T     LD 1;
      TAK;
      T     LD 5;
      L     #IN_TIMER_500MS_2;
      T     LW 9;
      L     LD 5;
      L     LD 1;
      A     T [LW 9];
      );
      JNB   _015;
      L     4;
      T     #STATUS;
_015: NOP   0;
NETWORK
TITLE = BOSALTIM VALFI CIKISI - NORMALDE ACIK
//1- Adim 1,2 ve 3 te bosaltim valfini kapat
//2- Adim 0 ve 4 te bosaltim valfi acik olacak
      A(;
      A     I 1.7;
      A(;
      L     #STATUS;
      L     0;
      ==I;
      );
      O(;
      L     #STATUS;
      L     4;
      ==I;
      );
      O(;
      L     #STATUS;
      L     5;
      ==I;
      );
      );
      AN    #IN_DIGER_KAZAN_BOSALTIMD;
      =     #ST_OUT_BOSALTIM_MEM;
NETWORK
TITLE = Adim 4 - Bosaltim Adimi
      L     #STATUS;
      L     4;
      ==I;
      =     L 0.0;
      A     L 0.0;
      JNB   _016;
      L     0.000000e+00;
      T     #ST_OUT_PID_MAN;
_016: NOP   0;
      A     L 0.0;
      BLD   102;
      =     #ST_KAZAN_BOSALTIMDA;
      A     L 0.0;
      A(;
      L     #O_SCALE_BASINC_OUT;
      L     1.000000e-01;
      <=R;
      );
      =     L 0.1;
      A     L 0.1;
      BLD   102;
      S     #st_OUT_adim4_emnyet_val;
      A(;
      A     L 0.1;
      L     S5T#5S;
      T     LD 1;
      TAK;
      T     LD 5;
      L     #IN_DELAY_BITISI_BEKLE;
      T     LW 9;
      L     LD 5;
      L     LD 1;
      SD    T [LW 9];
      NOP   0;
      NOP   0;
      NOP   0;
      T     LD 1;
      TAK;
      T     LD 5;
      L     #IN_DELAY_BITISI_BEKLE;
      T     LW 9;
      L     LD 5;
      L     LD 1;
      A     T [LW 9];
      );
      JNB   _017;
      L     5;
      T     #STATUS;
_017: NOP   0;
NETWORK
TITLE = KAPAK AÇILMASINI BEKLE
      A(;
      A(;
      L     #STATUS;
      L     5;
      ==I;
      );
      L     S5T#1S;
      T     LD 0;
      TAK;
      T     LD 4;
      L     #IN_DELAY_BIRAZ_BEKLE;
      T     LW 8;
      L     LD 4;
      L     LD 0;
      SD    T [LW 8];
      NOP   0;
      NOP   0;
      NOP   0;
      T     LD 0;
      TAK;
      T     LD 4;
      L     #IN_DELAY_BIRAZ_BEKLE;
      T     LW 8;
      L     LD 4;
      L     LD 0;
      A     T [LW 8];
      );
      AN    #IN_KAPAK;
      JNB   _018;
      L     0;
      T     #STATUS;
_018: NOP   0;
NETWORK
TITLE =
      AN    #IN_KAPAK;
      R     #st_OUT_adim4_emnyet_val;
NETWORK
TITLE =
//1- Acil Stop ile 1,2 ve 3. adimda ise bosaltim adimina git 
//2- 3. adimda bosalt butonu ile bosaltim yapabilsin  
      A(;
      AN    #IN_ACIL_STOP;
      A(;
      L     #STATUS;
      L     0;
      <>I;
      );
      A(;
      L     #STATUS;
      L     4;
      <>I;
      );
      A(;
      L     #STATUS;
      L     5;
      <>I;
      );
      O;
      A     #IN_BOSALTIM;
      A(;
      L     #STATUS;
      L     3;
      ==I;
      );
      );
      JNB   _019;
      L     4;
      T     #STATUS;
_019: NOP   0;
NETWORK
TITLE =
      A     I 1.6;
      JNB   _01a;
      L     0;
      T     #STATUS;
_01a: NOP   0;
NETWORK
TITLE = YESIL LAMBA
      A(;
      A     DB1.DBX 48.0;
      AN    #ST_PROSES_BASLADI;
      O(;
      L     #STATUS;
      L     5;
      ==I;
      );
      );
      A     I 1.7;
      A     M 0.5;
      =     #O_YESIL_LAM;
NETWORK
TITLE = KIRMIZI LAMBA
      A(;
      A     DB1.DBX 48.0;
      AN    #ST_PROSES_BASLADI;
      O(;
      L     #STATUS;
      L     1;
      ==I;
      );
      );
      A     I 1.7;
      A     M 0.5;
      =     #O_KIRMIZI_LAM;
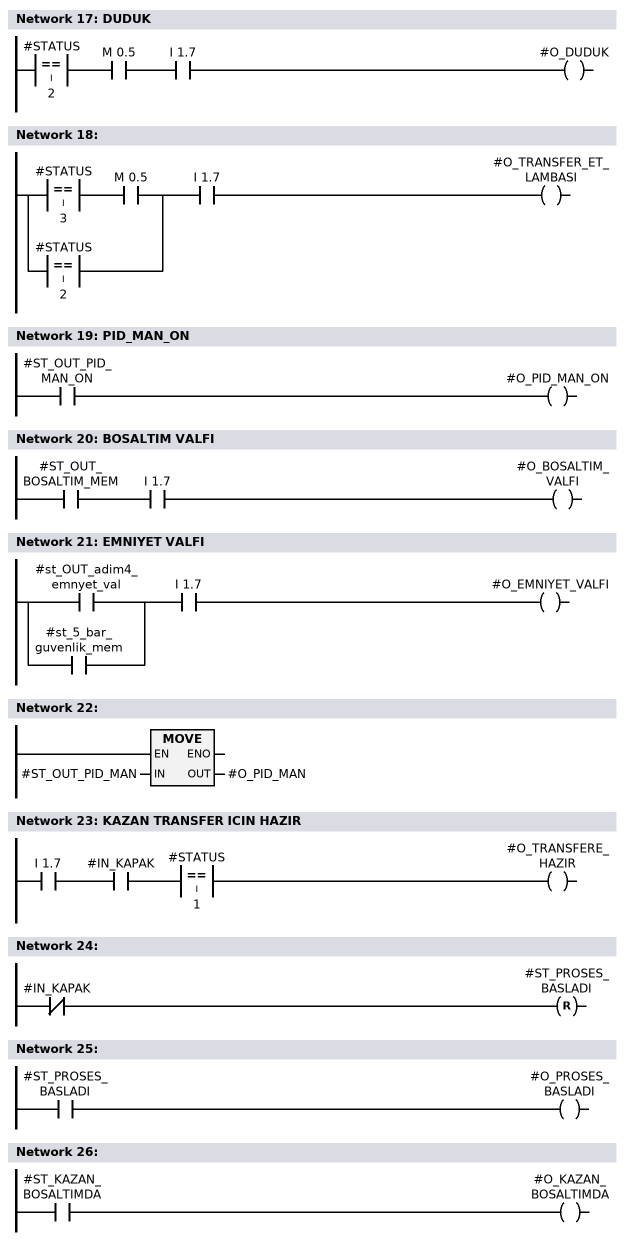
NETWORK
TITLE = DUDUK
      A(;
      L     #STATUS;
      L     2;
      ==I;
      );
      A     M 0.5;
      A     I 1.7;
      =     #O_DUDUK;
NETWORK
TITLE =
      A(;
      A(;
      L     #STATUS;
      L     3;
      ==I;
      );
      A     M 0.5;
      O(;
      L     #STATUS;
      L     2;
      ==I;
      );
      );
      A     I 1.7;
      =     #O_TRANSFER_ET_LAMBASI;
NETWORK
TITLE = PID_MAN_ON 
      A     #ST_OUT_PID_MAN_ON;
      =     #O_PID_MAN_ON;
NETWORK
TITLE = BOSALTIM VALFI
      A     #ST_OUT_BOSALTIM_MEM;
      A     I 1.7;
      =     #O_BOSALTIM_VALFI;
NETWORK
TITLE = EMNIYET VALFI
      A(;
      O     #st_OUT_adim4_emnyet_val;
      O     #st_5_bar_guvenlik_mem;
      );
      A     I 1.7;
      =     #O_EMNIYET_VALFI;
NETWORK
TITLE =
      L     #ST_OUT_PID_MAN;
      T     #O_PID_MAN;
      NOP   0;
NETWORK
TITLE = KAZAN TRANSFER ICIN HAZIR
      A     I 1.7;
      A     #IN_KAPAK;
      A(;
      L     #STATUS;
      L     1;
      ==I;
      );
      =     #O_TRANSFERE_HAZIR;
NETWORK
TITLE =
      AN    #IN_KAPAK;
      R     #ST_PROSES_BASLADI;
NETWORK
TITLE =
      A     #ST_PROSES_BASLADI;
      =     #O_PROSES_BASLADI;
NETWORK
TITLE =
      A     #ST_KAZAN_BOSALTIMDA;
      =     #O_KAZAN_BOSALTIMDA;
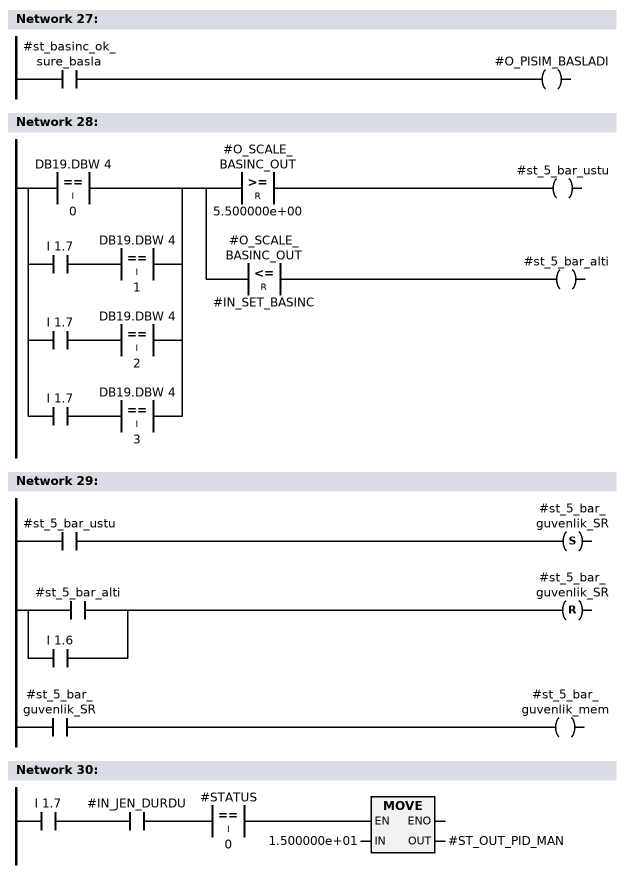
NETWORK
TITLE =
      A     #st_basinc_ok_sure_basla;
      =     #O_PISIM_BASLADI;
NETWORK
TITLE =
//Otoklav 5.5 bar'a geldiginde emniyet vantilini ac ve sete düþtügünde tekrar 
//emniyet ventilini kapat 
      O(;
      L     DB19.DBW 4;
      L     0;
      ==I;
      );
      O;
      A     I 1.7;
      A(;
      L     DB19.DBW 4;
      L     1;
      ==I;
      );
      O;
      A     I 1.7;
      A(;
      L     DB19.DBW 4;
      L     2;
      ==I;
      );
      O;
      A     I 1.7;
      A(;
      L     DB19.DBW 4;
      L     3;
      ==I;
      );
      =     L 0.0;
      A     L 0.0;
      A(;
      L     #O_SCALE_BASINC_OUT;
      L     5.500000e+00;
      >=R;
      );
      =     #st_5_bar_ustu;
      A     L 0.0;
      A(;
      L     #O_SCALE_BASINC_OUT;
      L     #IN_SET_BASINC;
      <=R;
      );
      =     #st_5_bar_alti;
NETWORK
TITLE =
      A     #st_5_bar_ustu;
      S     #st_5_bar_guvenlik_SR;
      A(;
      O     #st_5_bar_alti;
      O     I 1.6;
      );
      R     #st_5_bar_guvenlik_SR;
      A     #st_5_bar_guvenlik_SR;
      =     #st_5_bar_guvenlik_mem;
NETWORK
TITLE =
//JENERATORLER DURDUGUNDA BELIRLI SANIYE ORANSAL VANAYI AC HATTA BULUNAN BUHAR 
//TASFIYE EDILSIN
      A     I 1.7;
      A     #IN_JEN_DURDU;
      A(;
      L     #STATUS;
      L     0;
      ==I;
      );
      JNB   _01b;
      L     1.500000e+01;
      T     #ST_OUT_PID_MAN;
_01b: NOP   0;
END_FUNCTION_BLOCK

// FB 41: know-how protected block, not included

FUNCTION_BLOCK FB 47
//KAZAN 1 PID BLOGU
VERSION : 0.1
BEGIN
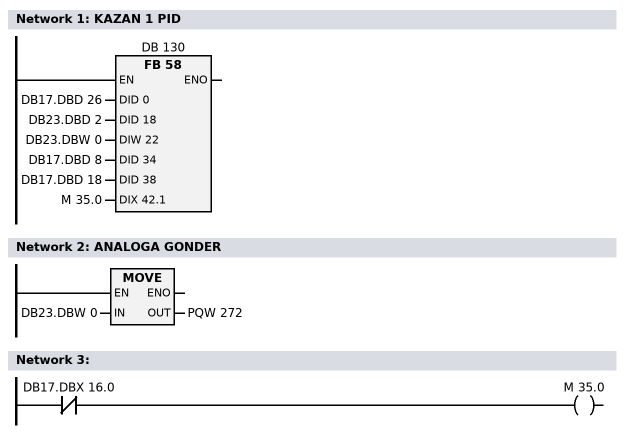
NETWORK
TITLE = KAZAN 1 PID
      CALL  FB 58 , DB 130 (
           DID 0                    := DB17.DBD 26,
           DID 18                   := DB23.DBD 2,
           DIW 22                   := DB23.DBW 0,
           DID 34                   := DB17.DBD 8,
           DID 38                   := DB17.DBD 18,
           DIX 42.1                 := M 35.0);
      NOP   0;
NETWORK
TITLE = ANALOGA GONDER
      L     DB23.DBW 0;
      T     PQW 272;
      NOP   0;
NETWORK
TITLE =
      AN    DB17.DBX 16.0;
      =     M 35.0;
NETWORK
TITLE =
END_FUNCTION_BLOCK

FUNCTION_BLOCK FB 48
VERSION : 0.1
BEGIN
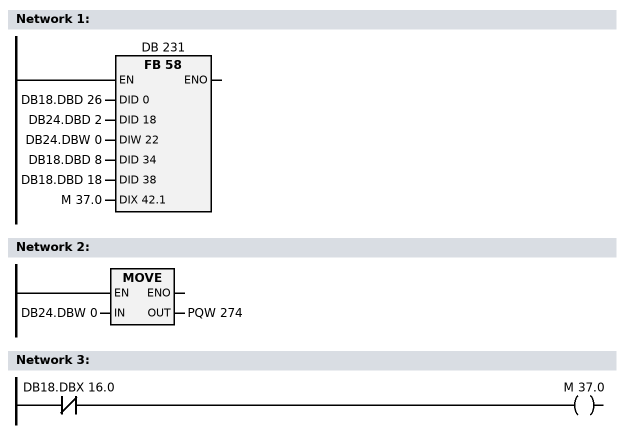
NETWORK
TITLE =
      CALL  FB 58 , DB 231 (
           DID 0                    := DB18.DBD 26,
           DID 18                   := DB24.DBD 2,
           DIW 22                   := DB24.DBW 0,
           DID 34                   := DB18.DBD 8,
           DID 38                   := DB18.DBD 18,
           DIX 42.1                 := M 37.0);
      NOP   0;
NETWORK
TITLE =
      L     DB24.DBW 0;
      T     PQW 274;
      NOP   0;
NETWORK
TITLE =
      AN    DB18.DBX 16.0;
      =     M 37.0;
END_FUNCTION_BLOCK

FUNCTION_BLOCK FB 49
//GAIN: 8.21488
//TI : 2.11452
//TD : 0.585774
//DERIVATIVE FACTOR: 5
//UPPER LIMIT : 80
//FACTOR : -1
//OFFSET : 100
VERSION : 0.1
VAR
  TCONT_C_MAN : REAL ;
  TCONT_C_MAN_ON : BOOL ;
  TCONT_C_LMN : REAL ;
  TCONT_C_LMN_PER : INT ;
END_VAR
BEGIN
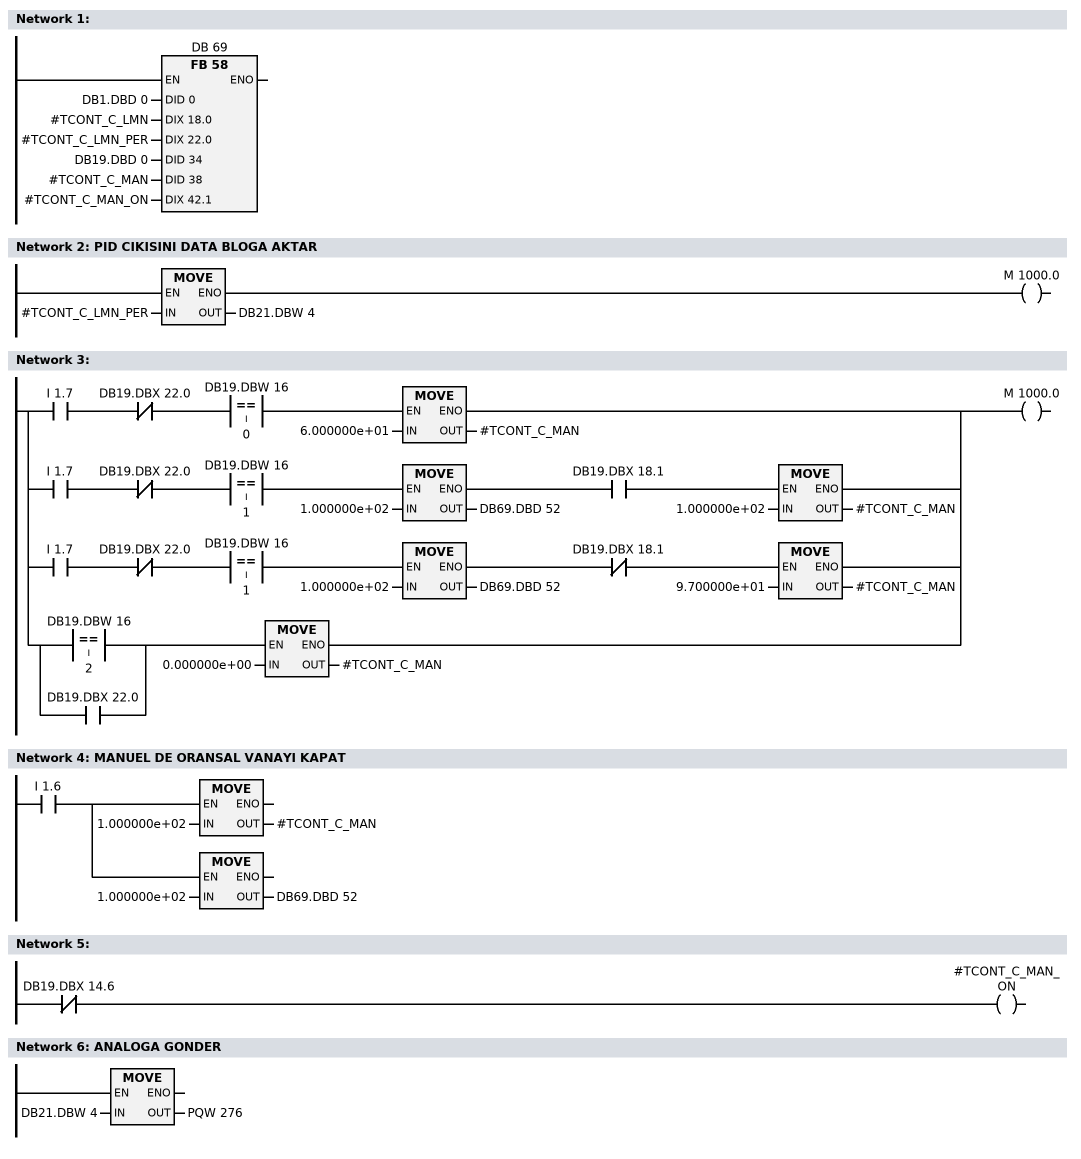
NETWORK
TITLE =
      CALL  FB 58 , DB 69 (
           DID 0                    := DB1.DBD 0,
           DIX 18.0                 := #TCONT_C_LMN,
           DIX 22.0                 := #TCONT_C_LMN_PER,
           DID 34                   := DB19.DBD 0,
           DID 38                   := #TCONT_C_MAN,
           DIX 42.1                 := #TCONT_C_MAN_ON);
      NOP   0;
NETWORK
TITLE = PID CIKISINI DATA BLOGA AKTAR
//SICAKLIK_2_OK  KISMINDAN PQW278 SILINDI. YERINE DB20.DBD0 BASINC SET DEGERI
//EKLENDI
      L     #TCONT_C_LMN_PER;
      T     DB21.DBW 4;
      SET;
      SAVE;
      CLR;
      A     BR;
      =     M 1000.0;
NETWORK
TITLE =
//FAZ DURUMUNA GORE MAN DEGERINI AYARLA
//FAZ 1 - MAN CIKIS OLARAK 40 GONDER- 40 TAN BASLAMASI ICIN
//FAZ 2 - TAMAMEN KAPANMASI ICIN 0 GONDER (PID MAUELDE)
//FAZ 3 - GUVENLIK SORUNLARINDA VANAYI TAMAMEN AC
      O(;
      A     I 1.7;
      AN    DB19.DBX 22.0;
      A(;
      L     DB19.DBW 16;
      L     0;
      ==I;
      );
      JNB   _001;
      L     6.000000e+01;
      T     #TCONT_C_MAN;
      SET;
      SAVE;
      CLR;
_001: A     BR;
      );
      O(;
      A(;
      A     I 1.7;
      AN    DB19.DBX 22.0;
      A(;
      L     DB19.DBW 16;
      L     1;
      ==I;
      );
      JNB   _002;
      L     1.000000e+02;
      T     DB69.DBD 52;
      SET;
      SAVE;
      CLR;
_002: A     BR;
      );
      A     DB19.DBX 18.1;
      JNB   _003;
      L     1.000000e+02;
      T     #TCONT_C_MAN;
      SET;
      SAVE;
      CLR;
_003: A     BR;
      );
      O(;
      A(;
      A     I 1.7;
      AN    DB19.DBX 22.0;
      A(;
      L     DB19.DBW 16;
      L     1;
      ==I;
      );
      JNB   _004;
      L     1.000000e+02;
      T     DB69.DBD 52;
      SET;
      SAVE;
      CLR;
_004: A     BR;
      );
      AN    DB19.DBX 18.1;
      JNB   _005;
      L     9.700000e+01;
      T     #TCONT_C_MAN;
      SET;
      SAVE;
      CLR;
_005: A     BR;
      );
      O(;
      A(;
      O(;
      L     DB19.DBW 16;
      L     2;
      ==I;
      );
      O     DB19.DBX 22.0;
      );
      JNB   _006;
      L     0.000000e+00;
      T     #TCONT_C_MAN;
      SET;
      SAVE;
      CLR;
_006: A     BR;
      );
      =     M 1000.0;
NETWORK
TITLE = MANUEL DE ORANSAL VANAYI KAPAT
      A     I 1.6;
      =     L 0.0;
      A     L 0.0;
      JNB   _007;
      L     1.000000e+02;
      T     #TCONT_C_MAN;
_007: NOP   0;
      A     L 0.0;
      JNB   _008;
      L     1.000000e+02;
      T     DB69.DBD 52;
_008: NOP   0;
NETWORK
TITLE =
      AN    DB19.DBX 14.6;
      =     #TCONT_C_MAN_ON;
NETWORK
TITLE = ANALOGA GONDER
      L     DB21.DBW 4;
      T     PQW 276;
      NOP   0;
END_FUNCTION_BLOCK

FUNCTION_BLOCK FB 50
//GAIN: 8.21488
//TI : 2.11452
//TD : 0.585774
//DERIVATIVE FACTOR: 5
//UPPER LIMIT : 80
//FACTOR : -1
//OFFSET : 100
VERSION : 0.1
VAR
  TCONT_C_LMN : REAL ;
  TCONT_C_LMN_PER : INT ;
  TCONT_C_MAN : REAL ;
  TCONT_C_MAN_ON : BOOL ;
  Ris_5_Bar : BOOL ;
END_VAR
BEGIN
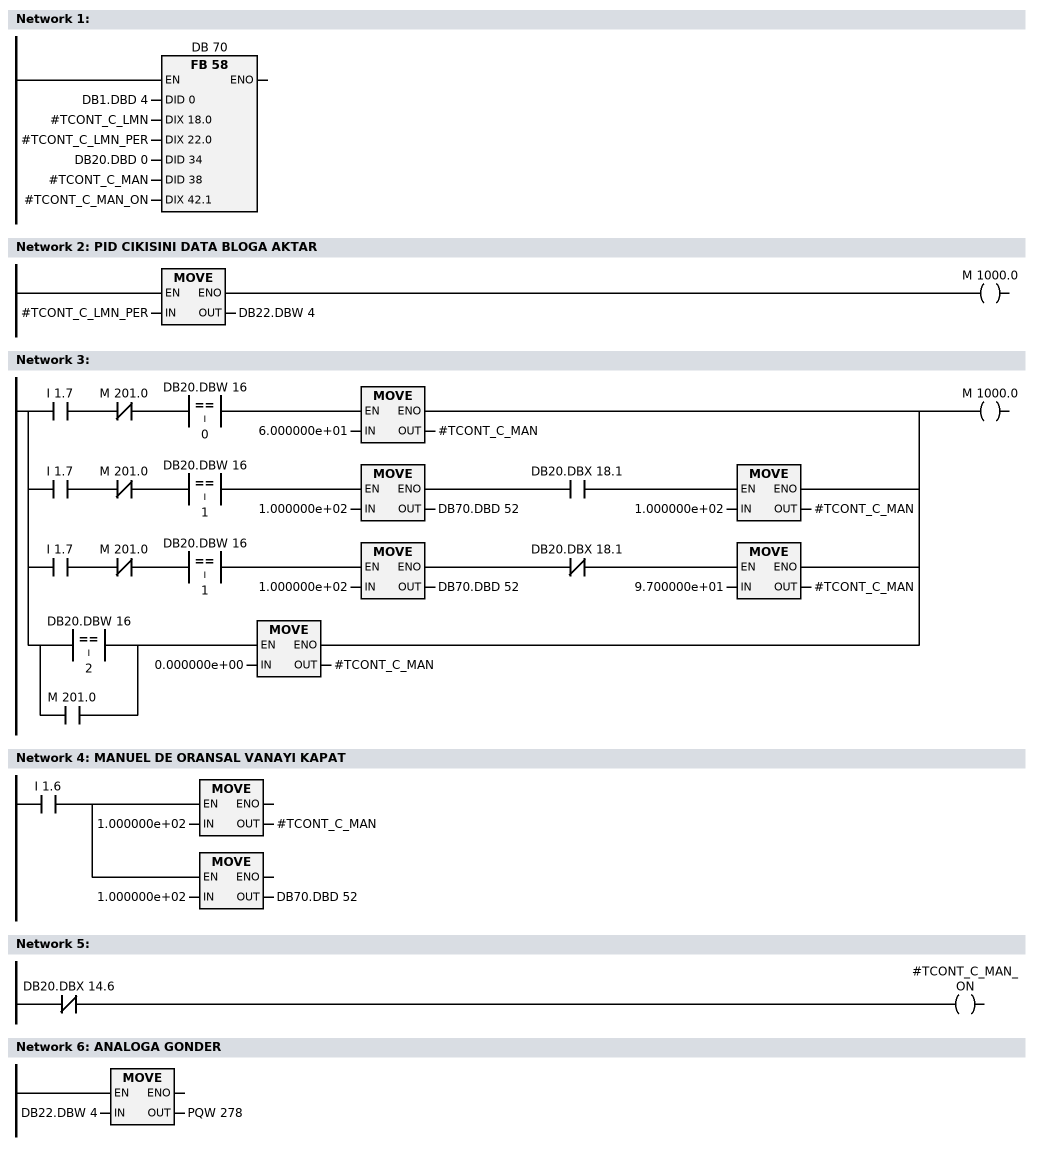
NETWORK
TITLE =
      CALL  FB 58 , DB 70 (
           DID 0                    := DB1.DBD 4,
           DIX 18.0                 := #TCONT_C_LMN,
           DIX 22.0                 := #TCONT_C_LMN_PER,
           DID 34                   := DB20.DBD 0,
           DID 38                   := #TCONT_C_MAN,
           DIX 42.1                 := #TCONT_C_MAN_ON);
      NOP   0;
NETWORK
TITLE = PID CIKISINI DATA BLOGA AKTAR
//SICAKLIK_2_OK  KISMINDAN PQW278 SILINDI. YERINE DB20.DBD0 BASINC SET DEGERI
//EKLENDI
      L     #TCONT_C_LMN_PER;
      T     DB22.DBW 4;
      SET;
      SAVE;
      CLR;
      A     BR;
      =     M 1000.0;
NETWORK
TITLE =
//FAZ DURUMUNA GORE MAN DEGERINI AYARLA
//FAZ 1 - MAN CIKIS OLARAK 40 GONDER- 40 TAN BASLAMASI ICIN
//FAZ 2 - TAMAMEN KAPANMASI ICIN 0 GONDER (PID MAUELDE)
//FAZ 3 - GUVENLIK SORUNLARINDA VANAYI TAMAMEN AC
      O(;
      A     I 1.7;
      AN    M 201.0;
      A(;
      L     DB20.DBW 16;
      L     0;
      ==I;
      );
      JNB   _001;
      L     6.000000e+01;
      T     #TCONT_C_MAN;
      SET;
      SAVE;
      CLR;
_001: A     BR;
      );
      O(;
      A(;
      A     I 1.7;
      AN    M 201.0;
      A(;
      L     DB20.DBW 16;
      L     1;
      ==I;
      );
      JNB   _002;
      L     1.000000e+02;
      T     DB70.DBD 52;
      SET;
      SAVE;
      CLR;
_002: A     BR;
      );
      A     DB20.DBX 18.1;
      JNB   _003;
      L     1.000000e+02;
      T     #TCONT_C_MAN;
      SET;
      SAVE;
      CLR;
_003: A     BR;
      );
      O(;
      A(;
      A     I 1.7;
      AN    M 201.0;
      A(;
      L     DB20.DBW 16;
      L     1;
      ==I;
      );
      JNB   _004;
      L     1.000000e+02;
      T     DB70.DBD 52;
      SET;
      SAVE;
      CLR;
_004: A     BR;
      );
      AN    DB20.DBX 18.1;
      JNB   _005;
      L     9.700000e+01;
      T     #TCONT_C_MAN;
      SET;
      SAVE;
      CLR;
_005: A     BR;
      );
      O(;
      A(;
      O(;
      L     DB20.DBW 16;
      L     2;
      ==I;
      );
      O     M 201.0;
      );
      JNB   _006;
      L     0.000000e+00;
      T     #TCONT_C_MAN;
      SET;
      SAVE;
      CLR;
_006: A     BR;
      );
      =     M 1000.0;
NETWORK
TITLE = MANUEL DE ORANSAL VANAYI KAPAT
      A     I 1.6;
      =     L 0.0;
      A     L 0.0;
      JNB   _007;
      L     1.000000e+02;
      T     #TCONT_C_MAN;
_007: NOP   0;
      A     L 0.0;
      JNB   _008;
      L     1.000000e+02;
      T     DB70.DBD 52;
_008: NOP   0;
NETWORK
TITLE =
      AN    DB20.DBX 14.6;
      =     #TCONT_C_MAN_ON;
NETWORK
TITLE = ANALOGA GONDER
      L     DB22.DBW 4;
      T     PQW 278;
      NOP   0;
END_FUNCTION_BLOCK

// FB 58: know-how protected block, not included

FUNCTION_BLOCK FB 94
VERSION : 0.1
BEGIN
NETWORK
TITLE =
      CALL  FB 20 , DB 120 (
           IN_ACIL_STOP             := I 0.0,
           IN_START                 := I 0.1,
           IN_TRANSFER              := I 0.2,
           IN_BOSALTIM              := I 0.3,
           IN_KAPAK                 := I 0.4,
           IN_JENS_OK               := DB17.DBX 2.0,
           IN_TRANSFERE_HAZIR       := DB17.DBX 2.1,
           IN_PISIM_SURESI          := DB17.DBW 4,
           IN_SCALE_BASINC_PER      := DB17.DBW 6,
           IN_SET_BASINC            := DB17.DBD 8,
           IN_DIGER_KAZAN_BASINCI   := DB17.DBD 12,
           IN_TIMER_500MS           := T 10,
           IN_TIMER_1S              := T 11,
           IN_TIMER_PISIRME         := T 12,
           IN_TIMER_500MS_2         := T 13,
           IN_TIMER_7S              := T 14,
           IN_SCALE_HI_LIM          := 1.000000e+01,
           IN_SCALE_LO_LIM          := 0.000000e+00,
           IN_SCALE_SICAKLIK_HI_LIM := 2.000000e+02,
           IN_SCALE_SICAKLIK_LO_LIM := 0.000000e+00,
           IN_SCALE_SICAKLIK_PER    := DB17.DBW 38,
           IN_DIGER_KAZAN_BOSALTIMD := DB17.DBX 40.1,
           IN_TRANSFER_BASLADI      := DB17.DBX 40.2,
           IN_JEN_DURDU             := DB2.DBX 16.0,
           IN_DELAY_BITISI_BEKLE    := T 51,
           IN_DELAY_BIRAZ_BEKLE     := T 52,
           O_YESIL_LAM              := Q 0.0,
           O_KIRMIZI_LAM            := Q 0.1,
           O_DUDUK                  := Q 0.2,
           O_BOSALTIM_VALFI         := Q 0.3,
           O_PID_MAN_ON             := DB17.DBX 16.0,
           O_PID_MAN                := DB17.DBD 18,
           O_TRANSFER_YAPILIYOR     := DB17.DBX 22.0,
           O_SCALE_BASINC_RET_VAL   := DB17.DBW 24,
           O_SCALE_BASINC_OUT       := DB17.DBD 26,
           O_EMNIYET_VALFI          := Q 0.5,
           O_TRANSFERE_HAZIR        := DB17.DBX 30.0,
           O_SCALE_SICAKLIK_RET_VAL := DB17.DBW 32,
           O_SCALE_SICAKLIK_OUT     := DB17.DBD 34,
           O_TRANSFER_ET_LAMBASI    := Q 0.4,
           O_PROSES_BASLADI         := M 300.0,
           O_KAZAN_BOSALTIMDA       := DB17.DBX 40.0,
           O_PISIM_BASLADI          := DB17.DBX 40.3,
           STATUS                   := DB17.DBW 0);
//       O_YESIL_LAM             :="KAZAN1_YESIL_LAMBA"
//       O_KIRMIZI_LAM           :="KAZAN1_KIRMIZI_LAMBA"
//       O_DUDUK                 :="KAZAN1_DUDUK"
//       O_BOSALTIM_VALFI        :="KAZAN1_BOSALTIM_VALFI"
//       O_PID_MAN_ON            :="KAZAN1_DATA".O_PID_MAN_ON
//       O_PID_MAN               :="KAZAN1_DATA".O_PID_MAN
//       O_TRANSFER_YAPILIYOR    :="KAZAN1_DATA".O_TRANSFER_YAPILIYOR
//       O_SCALE_BASINC_RET_VAL  :="KAZAN1_DATA".O_SCALE_BASINC_RET_VAL
//       O_SCALE_BASINC_OUT      :="KAZAN1_DATA".O_SCALE_BASINC_OUT
//       O_EMNIYET_VALFI         :="KAZAN1_EMN_VALFI_BOS"
//       O_TRANSFERE_HAZIR       :="KAZAN1_DATA".O_TRANSFERE_HAZIR
//       O_SCALE_SICAKLIK_RET_VAL:="KAZAN1_DATA".O_SCALE_SICAKLIK_RET_VAL
//       O_SCALE_SICAKLIK_OUT    :="KAZAN1_DATA".O_SCALE_SICAKLIK_OUT
//       O_TRANSFER_ET_LAMBASI   :="KAZAN1_TRANS_BUT_LAMBASI"
//       O_PROSES_BASLADI        :=M300.0
//       O_KAZAN_BOSALTIMDA      :="KAZAN1_DATA".O_KAZAN_BOSALTIMDA
//       O_PISIM_BASLADI         :="KAZAN1_DATA".O_PISIM_BASLADI
//       STATUS                  :="KAZAN1_DATA".IN_STATUS
NETWORK
TITLE = GIRIS-CIKIS
      A     DB18.DBX 30.0;
      =     DB17.DBX 2.1;
      L     PIW 272;
      T     DB17.DBW 6;
      L     PIW 274;
      T     DB17.DBW 38;
      L     DB18.DBD 26;
      T     DB17.DBD 12;
      O     DB19.DBX 18.2;
      O     DB20.DBX 18.2;
      =     DB17.DBX 2.0;
      A     DB18.DBX 40.0;
      =     DB17.DBX 40.1;
      A     DB18.DBX 22.0;
      =     DB17.DBX 40.2;
END_FUNCTION_BLOCK

FUNCTION_BLOCK FB 95
VERSION : 0.1
BEGIN
NETWORK
TITLE =
      CALL  FB 20 , DB 230 (
           IN_ACIL_STOP             := I 0.5,
           IN_START                 := I 0.6,
           IN_TRANSFER              := I 0.7,
           IN_BOSALTIM              := I 1.0,
           IN_KAPAK                 := I 1.1,
           IN_JENS_OK               := DB18.DBX 2.0,
           IN_TRANSFERE_HAZIR       := DB18.DBX 2.1,
           IN_PISIM_SURESI          := DB18.DBW 4,
           IN_SCALE_BASINC_PER      := DB18.DBW 6,
           IN_SET_BASINC            := DB18.DBD 8,
           IN_DIGER_KAZAN_BASINCI   := DB18.DBD 12,
           IN_TIMER_500MS           := T 20,
           IN_TIMER_1S              := T 21,
           IN_TIMER_PISIRME         := T 22,
           IN_TIMER_500MS_2         := T 23,
           IN_TIMER_7S              := T 24,
           IN_SCALE_HI_LIM          := 1.000000e+01,
           IN_SCALE_LO_LIM          := 0.000000e+00,
           IN_SCALE_SICAKLIK_HI_LIM := 2.000000e+02,
           IN_SCALE_SICAKLIK_LO_LIM := 0.000000e+00,
           IN_SCALE_SICAKLIK_PER    := DB18.DBW 38,
           IN_DIGER_KAZAN_BOSALTIMD := DB18.DBX 40.1,
           IN_TRANSFER_BASLADI      := DB18.DBX 40.2,
           IN_JEN_DURDU             := DB2.DBX 16.0,
           IN_DELAY_BITISI_BEKLE    := T 50,
           IN_DELAY_BIRAZ_BEKLE     := T 53,
           O_YESIL_LAM              := Q 0.6,
           O_KIRMIZI_LAM            := Q 0.7,
           O_DUDUK                  := Q 1.0,
           O_BOSALTIM_VALFI         := Q 1.1,
           O_PID_MAN_ON             := DB18.DBX 16.0,
           O_PID_MAN                := DB18.DBD 18,
           O_TRANSFER_YAPILIYOR     := DB18.DBX 22.0,
           O_SCALE_BASINC_RET_VAL   := DB18.DBW 24,
           O_SCALE_BASINC_OUT       := DB18.DBD 26,
           O_EMNIYET_VALFI          := Q 1.3,
           O_TRANSFERE_HAZIR        := DB18.DBX 30.0,
           O_SCALE_SICAKLIK_RET_VAL := DB18.DBW 32,
           O_SCALE_SICAKLIK_OUT     := DB18.DBD 34,
           O_TRANSFER_ET_LAMBASI    := Q 1.2,
           O_PROSES_BASLADI         := M 300.1,
           O_KAZAN_BOSALTIMDA       := DB18.DBX 40.0,
           O_PISIM_BASLADI          := DB18.DBX 40.3,
           STATUS                   := DB18.DBW 0);
//       O_YESIL_LAM             :="KAZAN2_YESIL_LAMBA"
//       O_KIRMIZI_LAM           :="KAZAN2_KIRMIZI_LAMBA"
//       O_DUDUK                 :="KAZAN2_DUDUK"
//       O_BOSALTIM_VALFI        :="KAZAN2_BOSALTIM_VALFI"
//       O_PID_MAN_ON            :="KAZAN2_DATA".O_PID_MAN_ON
//       O_PID_MAN               :="KAZAN2_DATA".O_PID_MAN
//       O_TRANSFER_YAPILIYOR    :="KAZAN2_DATA".O_TRANSFER_YAPILIYOR
//       O_SCALE_BASINC_RET_VAL  :="KAZAN2_DATA".O_SCALE_BASINC_RET_VAL
//       O_SCALE_BASINC_OUT      :="KAZAN2_DATA".O_SCALE_BASINC_OUT
//       O_EMNIYET_VALFI         :="KAZAN2_EMN_VALFI_BOS"
//       O_TRANSFERE_HAZIR       :="KAZAN2_DATA".O_TRANSFERE_HAZIR
//       O_SCALE_SICAKLIK_RET_VAL:="KAZAN2_DATA".O_SCALE_SICAKLIK_RET_VAL
//       O_SCALE_SICAKLIK_OUT    :="KAZAN2_DATA".O_SCALE_SICAKLIK_OUT
//       O_TRANSFER_ET_LAMBASI   :="KAZAN2_TRANS_BUT_LAMBASI"
//       O_PROSES_BASLADI        :=M300.1
//       O_KAZAN_BOSALTIMDA      :="KAZAN2_DATA".O_KAZAN_BOSALTIMDA
//       O_PISIM_BASLADI         :="KAZAN2_DATA".O_PISIM_BASLADI
//       STATUS                  :="KAZAN2_DATA".IN_STATUS
NETWORK
TITLE =
      A     DB17.DBX 30.0;
      =     DB18.DBX 2.1;
      L     PIW 276;
      T     DB18.DBW 6;
      L     PIW 278;
      T     DB18.DBW 38;
      L     DB17.DBD 26;
      T     DB18.DBD 12;
      O     DB19.DBX 18.2;
      O     DB20.DBX 18.2;
      =     DB18.DBX 2.0;
      A     DB17.DBX 40.0;
      =     DB18.DBX 40.1;
      A     DB17.DBX 22.0;
      =     DB18.DBX 40.2;
END_FUNCTION_BLOCK

FUNCTION_BLOCK FB 98
VERSION : 0.1
VAR
  st_Set_100_Derece : BOOL ;
  Set1_OK : BOOL ;
  st_Stop_Trigger : BOOL ;
  st_Stop_Set_Mem : BOOL ;
  st_Sicaklik_Dustu : BOOL ;
END_VAR
VAR_TEMP
  t_Ris_Set_100 : BOOL ;
  t_Ris_Start : BOOL ;
  t_Ris_Status : BOOL ;
  t_Ris_Status2 : BOOL ;
  t_Ris_Status3 : BOOL ;
  t_Ris_Set1_ok : BOOL ;
  t_Ris_Set1_ok_1 : BOOL ;
  t_Ris_Set1_ok_2 : BOOL ;
  t_Ris_Stop : BOOL ;
  t_Ris_Sogutma : BOOL ;
  t_Fall_Sogutma : BOOL ;
  t_Ris_Sicaklik_Dustu : BOOL ;
END_VAR
BEGIN
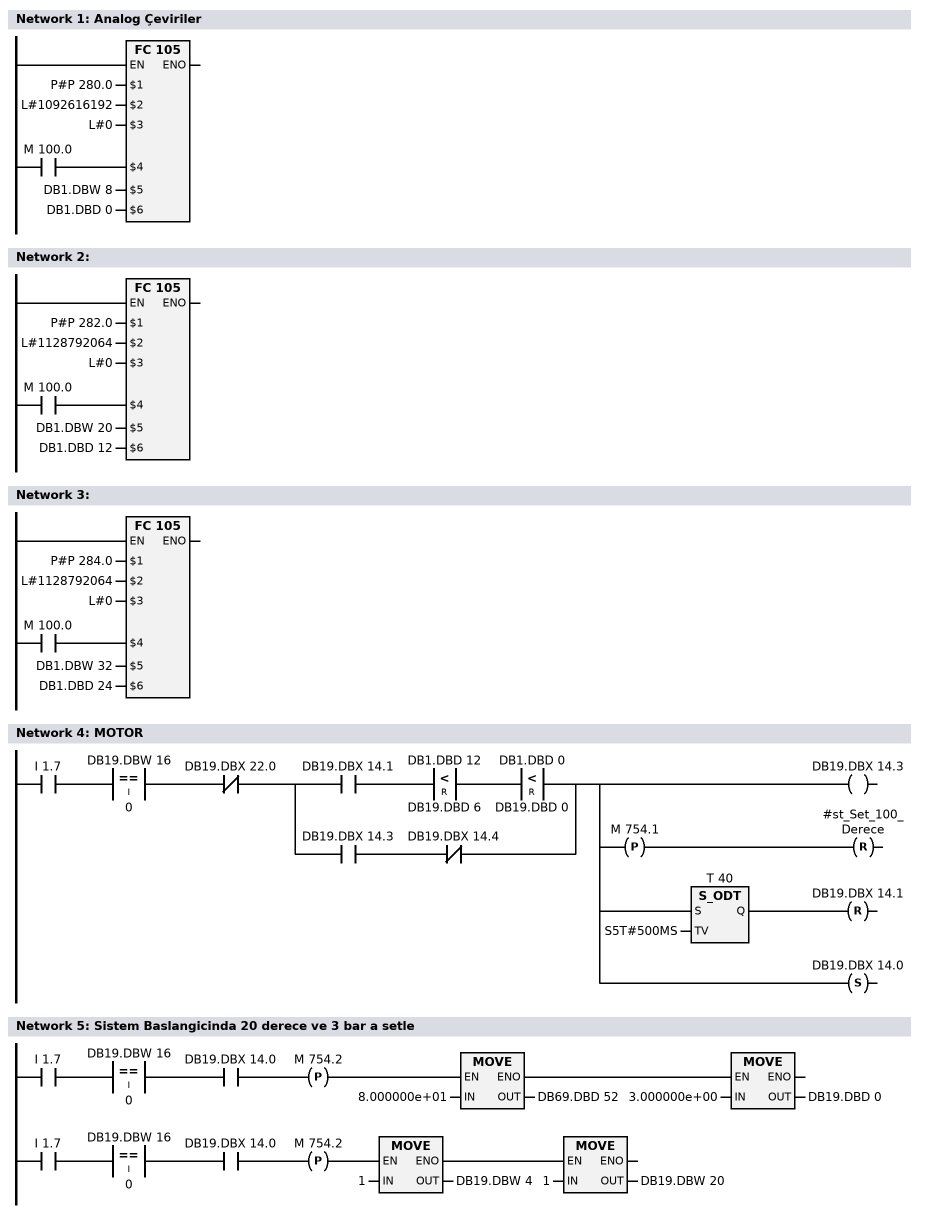
NETWORK
TITLE = Analog Çeviriler
      A     M 100.0;
      =     L 2.0;
      BLD   103;
      CALL  FC 105 (
           $1                       := P#P 280.0,
           $2                       := L#1092616192,
           $3                       := L#0,
           $4                       := L 2.0,
           $5                       := DB1.DBW 8,
           $6                       := DB1.DBD 0);
      NOP   0;
NETWORK
TITLE =
      A     M 100.0;
      =     L 2.0;
      BLD   103;
      CALL  FC 105 (
           $1                       := P#P 282.0,
           $2                       := L#1128792064,
           $3                       := L#0,
           $4                       := L 2.0,
           $5                       := DB1.DBW 20,
           $6                       := DB1.DBD 12);
      NOP   0;
NETWORK
TITLE =
      A     M 100.0;
      =     L 2.0;
      BLD   103;
      CALL  FC 105 (
           $1                       := P#P 284.0,
           $2                       := L#1128792064,
           $3                       := L#0,
           $4                       := L 2.0,
           $5                       := DB1.DBW 32,
           $6                       := DB1.DBD 24);
      NOP   0;
NETWORK
TITLE = MOTOR
      A     I 1.7;
      A(;
      L     DB19.DBW 16;
      L     0;
      ==I;
      );
      AN    DB19.DBX 22.0;
      A(;
      A     DB19.DBX 14.1;
      A(;
      L     DB1.DBD 12;
      L     DB19.DBD 6;
      <R;
      );
      A(;
      L     DB1.DBD 0;
      L     DB19.DBD 0;
      <R;
      );
      O;
      A     DB19.DBX 14.3;
      AN    DB19.DBX 14.4;
      );
      =     L 2.0;
      A     L 2.0;
      BLD   102;
      =     DB19.DBX 14.3;
      A     L 2.0;
      FP    M 754.1;
      R     #st_Set_100_Derece;
      A     L 2.0;
      L     S5T#500MS;
      SD    T 40;
      NOP   0;
      NOP   0;
      NOP   0;
      A     T 40;
      R     DB19.DBX 14.1;
      A     L 2.0;
      BLD   102;
      S     DB19.DBX 14.0;
NETWORK
TITLE = Sistem Baslangicinda 20 derece ve 3 bar a setle
      A     I 1.7;
      A(;
      L     DB19.DBW 16;
      L     0;
      ==I;
      );
      A     DB19.DBX 14.0;
      FP    M 754.2;
      =     L 2.0;
      A(;
      A     L 2.0;
      JNB   _001;
      L     8.000000e+01;
      T     DB69.DBD 52;
      SET;
      SAVE;
      CLR;
_001: A     BR;
      );
      JNB   _002;
      L     3.000000e+00;
      T     DB19.DBD 0;
_002: NOP   0;
      A(;
      A     L 2.0;
      JNB   _003;
      L     1;
      T     DB19.DBW 4;
      SET;
      SAVE;
      CLR;
_003: A     BR;
      );
      JNB   _004;
      L     1;
      T     DB19.DBW 20;
_004: NOP   0;
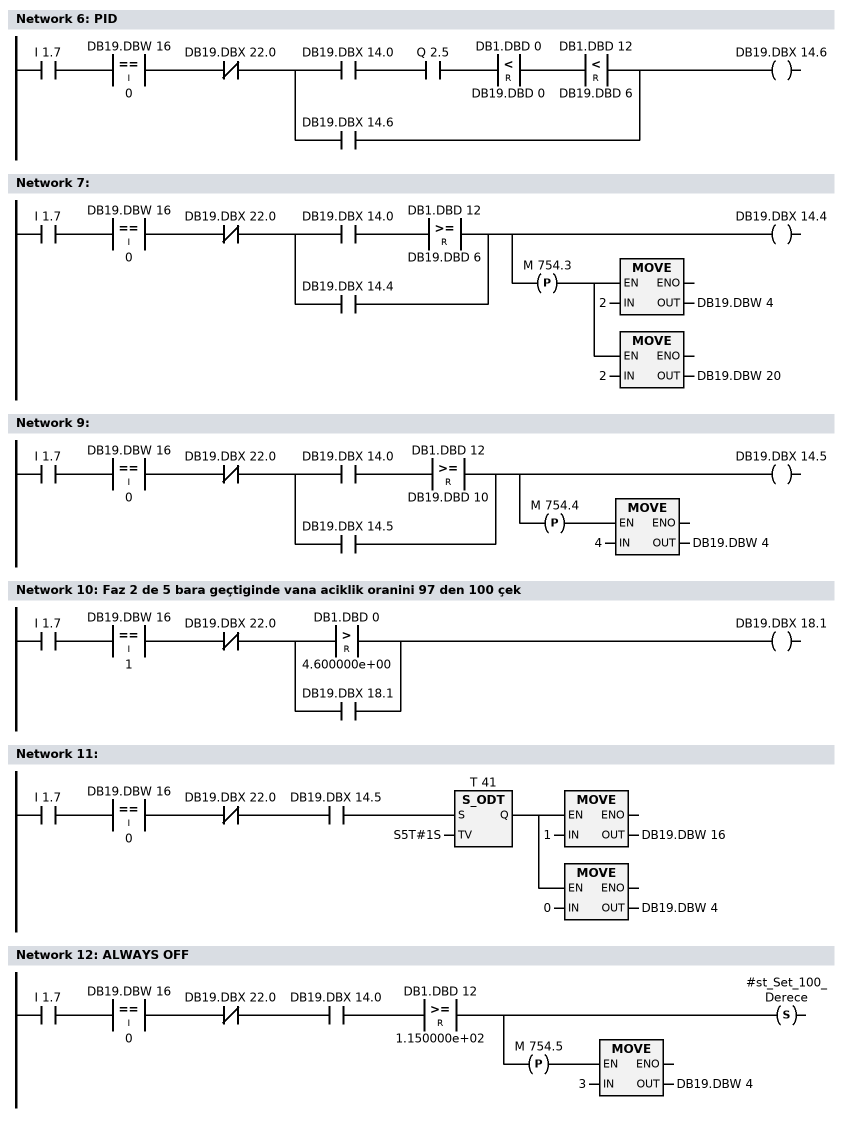
NETWORK
TITLE = PID
      A     I 1.7;
      A(;
      L     DB19.DBW 16;
      L     0;
      ==I;
      );
      AN    DB19.DBX 22.0;
      A(;
      A     DB19.DBX 14.0;
      A     Q 2.5;
      A(;
      L     DB1.DBD 0;
      L     DB19.DBD 0;
      <R;
      );
      A(;
      L     DB1.DBD 12;
      L     DB19.DBD 6;
      <R;
      );
      O     DB19.DBX 14.6;
      );
      =     DB19.DBX 14.6;
NETWORK
TITLE =
      A     I 1.7;
      A(;
      L     DB19.DBW 16;
      L     0;
      ==I;
      );
      AN    DB19.DBX 22.0;
      A(;
      A     DB19.DBX 14.0;
      A(;
      L     DB1.DBD 12;
      L     DB19.DBD 6;
      >=R;
      );
      O     DB19.DBX 14.4;
      );
      =     L 2.0;
      A     L 2.0;
      BLD   102;
      =     DB19.DBX 14.4;
      A     L 2.0;
      FP    M 754.3;
      =     L 2.1;
      A     L 2.1;
      JNB   _005;
      L     2;
      T     DB19.DBW 4;
_005: NOP   0;
      A     L 2.1;
      JNB   _006;
      L     2;
      T     DB19.DBW 20;
_006: NOP   0;
NETWORK
TITLE = SET 2 DEGERINE ULASMADI ISE BRULOR VE MOTORU CALISTIR
      A(;
      A     DB19.DBX 14.4;
      FP    M 101.1;
      S     M 101.0;
      A(;
      O(;
      L     DB19.DBW 16;
      L     1;
      ==I;
      );
      O     DB19.DBX 22.0;
      );
      R     M 101.0;
      A     M 101.0;
      );
      L     S5T#1M30S;
      SD    T 57;
      NOP   0;
      NOP   0;
      NOP   0;
      A     T 57;
      =     DB19.DBX 38.0;
NETWORK
TITLE =
      A     I 1.7;
      A(;
      L     DB19.DBW 16;
      L     0;
      ==I;
      );
      AN    DB19.DBX 22.0;
      A(;
      A     DB19.DBX 14.0;
      A(;
      L     DB1.DBD 12;
      L     DB19.DBD 10;
      >=R;
      );
      O     DB19.DBX 14.5;
      );
      =     L 2.0;
      A     L 2.0;
      BLD   102;
      =     DB19.DBX 14.5;
      A     L 2.0;
      FP    M 754.4;
      JNB   _007;
      L     4;
      T     DB19.DBW 4;
_007: NOP   0;
NETWORK
TITLE = Faz 2 de 5 bara geçtiginde vana aciklik oranini 97 den 100 çek
      A     I 1.7;
      A(;
      L     DB19.DBW 16;
      L     1;
      ==I;
      );
      AN    DB19.DBX 22.0;
      A(;
      O(;
      L     DB1.DBD 0;
      L     4.600000e+00;
      >R;
      );
      O     DB19.DBX 18.1;
      );
      =     DB19.DBX 18.1;
NETWORK
TITLE =
//SET 2 SICAKLIGINDAN SONRA FAZ 2 E GEC
      A     I 1.7;
      A(;
      L     DB19.DBW 16;
      L     0;
      ==I;
      );
      AN    DB19.DBX 22.0;
      A     DB19.DBX 14.5;
      L     S5T#1S;
      SD    T 41;
      NOP   0;
      NOP   0;
      NOP   0;
      A     T 41;
      =     L 2.0;
      A     L 2.0;
      JNB   _008;
      L     1;
      T     DB19.DBW 16;
_008: NOP   0;
      A     L 2.0;
      JNB   _009;
      L     0;
      T     DB19.DBW 4;
_009: NOP   0;
NETWORK
TITLE = ALWAYS OFF
//Pompa 100 derecede duracak
      A     I 1.7;
      A(;
      L     DB19.DBW 16;
      L     0;
      ==I;
      );
      AN    DB19.DBX 22.0;
      A     DB19.DBX 14.0;
      A(;
      L     DB1.DBD 12;
      L     1.150000e+02;
      >=R;
      );
      =     L 2.0;
      A     L 2.0;
      BLD   102;
      S     #st_Set_100_Derece;
      A     L 2.0;
      FP    M 754.5;
      JNB   _00a;
      L     3;
      T     DB19.DBW 4;
_00a: NOP   0;
